(******************************************************************************************************************************************)
(****************************				           Reset Function Part                                                 *****************************)
(******************************************************************************************************************************************)
IF xReset THEN
	xReset:=FALSE;
	xSetEnd:=TRUE;
END_IF;
(******************************************************************************************************************************************)
(****************************				              Error Controlling Part                                            *****************************)
(******************************************************************************************************************************************)
IF (xSetError OR T_Station.TControl.xError) AND NOT(xSetEnd) THEN
	IF NOT(xInitError) THEN
		iStepError:=100;
		xInitError:=TRUE;
		T_Station.TControl.iCountDownPlungeCycle:=1;
		IF NOT(xSetError) THEN
			xSetError:=TRUE;
			xSetTmpError:=FALSE;
		ELSE
			xSetTmpError:=TRUE;
		END_IF;
	END_IF;
	CASE iStepError OF
		100:	IF T_Station.TControl.xError THEN
				diErrorNr:=T_Station.TControl.diErrorNr;
			END_IF;
			IF xSetTmpError THEN
				diErrorNr:=diTmpErrNr;
			END_IF;
			iStepError:=200;
		200:	IF xSetTmpError THEN
				xSetTmpError:=FALSE;
				xStopFctStation1:=FALSE;
				iStepError:=300;
			ELSE
				IF NOT(T_Station.TControl.xError) AND NOT(T_Station.TControl.xEnd) THEN
					IF (T_Station.TControl.iFunctNr = 1) THEN
						T_Station.TControl.xStop:=TRUE;
						xStopFctStation1:=TRUE;
					ELSE
						xStopFctStation1:=FALSE;
					END_IF;
				END_IF;
				iStepError:=300;
			END_IF;
		300:	IF xStopFctStation1 THEN
				IF NOT(T_Station.TControl.xStop) THEN
					xStopFctStation1:=FALSE;
				END_IF;
			END_IF;
			IF NOT(xStopFctStation1) THEN
				xError:=TRUE;
				iStepError:=400;
			END_IF;
		400:	IF xQuitErr THEN
				T_Station.TControl.xQuitError:=T_Station.TControl.xError;
				iStepError:=500;
			END_IF;
		500: IF NOT(T_Station.TControl.xQuitError) THEN
				xSetEnd:=TRUE;
			END_IF;
	END_CASE;
END_IF;
(******************************************************************************************************************************************)
(****************************				              Main Controlling Part                                            *****************************)
(******************************************************************************************************************************************)
IF (xStart OR xStartMainCtr) AND NOT(xSetEnd) AND NOT(xSetError) THEN
	IF NOT (xInitMainCtr) THEN
		iStepPrc:=10;
		xInitMainCtr:=TRUE;
		xStartMainCtr:=TRUE;
		xStart:=FALSE;
		xEnd:=FALSE;
		xSetEndPrc:=FALSE;
		iTmpFunctionNr:=1;
		xAbord:=FALSE;
		xProcessHold:=FALSE;
		T_ExchgParam.T_InfoValueCommon.iCountDownCycle:=1;
		xDoNotMovePositionOfToolFeeder:=FALSE;
		T_ExchgParam.T_InfoValueCommon.rActualWireFeedPosition:=0.0;
		T_ExchgParam.T_InfoValueCommon.rActualWireFeedSpeed:=0.0;
		(*08.07.2014: KFS	{	*)
		xWarmUp:= xWarmUpCycle:= T_ExchgParam.T_StationCommon.T_AutoGeometryPara.xWarmUp;
		xWarmUpDone:=FALSE;
		(*08.07.2014: KFS	}	*)
	END_IF;
	IF (xStopCycle AND NOT(xTmpStopCycle)) THEN
		IF (T_NovRAMData.T_ProcessImageData.T_AutoGeometryPara.iCycleGeometry <= 1) THEN
			xStopCycle:=xProcessHold:=FALSE;
			RETURN;
		END_IF;
		IF (iStepPrc = 40) AND NOT(xInitStep) THEN
			xTmpStopCycle:=TRUE;
		END_IF;
	END_IF;
	IF xTmpStopCycle THEN
		xStopCycle:=FALSE;
		xProcessHold:=TRUE;
		xTmpStopCycle:=FALSE;
		xInitStep:=xStartMainPrc:=FALSE;
		(*08.07.2014: KFS	{	*)
		xWarmUp:=FALSE;
		(*08.07.2014: KFS	}	*)
		iStepPrc:=100;
		RETURN;
	END_IF;
	IF xStop AND NOT(xTmpStop) THEN
		xTmpStop:=TRUE;
		iStepStop:=1;
	END_IF;
	IF xTmpStop THEN
		CASE iStepStop OF
		1:	IF NOT(T_Station.TControl.xEnd) THEN
				T_Station.TControl.xStop:=TRUE;
				iStepStop:=10;
			ELSE
				iStepStop:=20;
			END_IF;
		10:	IF NOT(T_Station.TControl.xStop) THEN
				iStepStop:=20;
			END_IF;
		20:	IF NOT(T_Station.TControl.xStart) AND T_Station.TControl.xEnd THEN
				T_Station.TControl.iFunctNr:=4;
				T_Station.TControl.xStart:=TRUE;
				T_Station.THardware.TAxisGrindFeeder.T_CtrleSingle.lrAcceleration:=T_NovRAMData.T_Standard.T_TeachINGrindFeeder.rAcceleration;
				T_Station.THardware.TAxisGrindFeeder.T_CtrleSingle.lrDecceleration:=T_NovRAMData.T_Standard.T_TeachINGrindFeeder.rDeceleration;
				T_Station.THardware.TAxisGrindFeeder.T_CtrleSingle.lrPosition:=	T_NovRAMData.T_ProcessImageData.T_ProcessPara.rToolDiameterProcess +
																			T_NovRAMData.T_ProcessImageData.T_ProcessPara.rSecurityPosGrindFeedProcess;
				T_Station.THardware.TAxisGrindFeeder.T_CtrleSingle.lrVelocity:=T_NovRAMData.T_ProcessImageData.T_ProcessPara.rSpeedBackwardGrindFeed;
				iStepStop:=30;
			END_IF;
		(* Check Active Movement of the Axis *)
		30:	IF NOT(T_Station.TControl.xStart) AND T_Station.TControl.xEnd THEN
				T_Station.TControl.iFunctNr:=18;	(* Check Axis Movement, and stop it if moves *)
				T_Station.TControl.xStart:=TRUE;
				iStepStop:=40;
			END_IF;
		40:	IF NOT(T_Station.TControl.xStart) AND T_Station.TControl.xEnd THEN
(*08.07.2014: KFS	{	*)
				IF iStepPrc = 105 THEN
					T_Station.THardware.TCylToolTension.T_CtrleCyl.iFunction:=2;
					T_Station.THardware.TCylToolTension.T_CtrleCyl.T_AnalogCylinder.rForceIn:=T_NovRAMData.T_ProcessImageData.T_ProcessPara.rToolTensionProcess;
					T_Station.THardware.TCylToolTension.T_Config.tDelayOn:=T#1s;
					T_Station.THardware.TCylToolTension.T_CtrleCyl.xExecute:=TRUE;
					T_Station.THardware.TCylToolLeftActive.T_CtrleCyl.iFunction:= 1;
					T_Station.THardware.TCylToolLeftActive.T_CtrleCyl.xExecute:=TRUE;
					T_Station.THardware.TCylToolRightActive.T_CtrleCyl.iFunction:=1;
					T_Station.THardware.TCylToolRightActive.T_CtrleCyl.xExecute:=TRUE;
					T_Station.THardware.TCylToolCenterActive.T_CtrleCyl.iFunction:=1;
					T_Station.THardware.TCylToolCenterActive.T_CtrleCyl.xExecute:=TRUE;
					T_Station.THardware.TCylToolPrismaLeftActive.T_CtrleCyl.iFunction:=1;
					T_Station.THardware.TCylToolPrismaLeftActive.T_CtrleCyl.xExecute:=TRUE;
					T_Station.THardware.TCylToolPrismaRightActive.T_CtrleCyl.iFunction:=1;
					T_Station.THardware.TCylToolPrismaRightActive.T_CtrleCyl.xExecute:=TRUE;
					iStepStop:=45;
				ELSE
(*08.07.2014: KFS	}	*)
					xStartMainPrc:=FALSE;
					xInitStep:=FALSE;
					iStepPrc:=0;
					xSetEnd:=TRUE;
					RETURN;
				END_IF
			END_IF;
		45:IF    (NOT(T_Station.THardware.TCylToolTension.T_CtrleCyl.xExecute) AND T_Station.THardware.TCylToolTension.T_CtrleCyl.xDone ) AND
		             (NOT(T_Station.THardware.TCylToolLeftActive.T_CtrleCyl.xExecute) AND T_Station.THardware.TCylToolLeftActive.T_CtrleCyl.xDone ) AND
			    (NOT(T_Station.THardware.TCylToolRightActive.T_CtrleCyl.xExecute) AND T_Station.THardware.TCylToolRightActive.T_CtrleCyl.xDone ) AND
			    (NOT(T_Station.THardware.TCylToolCenterActive.T_CtrleCyl.xExecute) AND T_Station.THardware.TCylToolCenterActive.T_CtrleCyl.xDone ) AND
			    (NOT(T_Station.THardware.TCylToolPrismaLeftActive.T_CtrleCyl.xExecute) AND T_Station.THardware.TCylToolPrismaLeftActive.T_CtrleCyl.xDone ) AND
			    (NOT(T_Station.THardware.TCylToolPrismaRightActive.T_CtrleCyl.xExecute) AND T_Station.THardware.TCylToolPrismaRightActive.T_CtrleCyl.xDone )		THEN
				xStartMainPrc:=FALSE;
				xInitStep:=FALSE;
				iStepPrc:=0;
				xSetEnd:=TRUE;
				RETURN;
			END_IF;
		END_CASE;
		RETURN;
	END_IF;
	IF NOT(xStartMainPrc) THEN
		xStartMainPrc:=TRUE;
	END_IF;
END_IF;
(******************************************************************************************************************************************)
(****************************				             Main Procedure Part                                             *****************************)
(******************************************************************************************************************************************)
(*08.07.2014: KFS	{	*)
IF xWarmUp AND NOT(xWarmUpDone)THEN
	TONWarmUpTimer(IN:=TRUE,PT:=T#45m);
	IF TONWarmUpTimer.Q THEN
		TONWarmUpTimer(IN:=FALSE);
		xWarmUpDone:=TRUE;
	END_IF;
ELSE
	TONWarmUpTimer(IN:=FALSE);
END_IF;
(*08.07.2014: KFS	}	*)
IF xStartProcess THEN
	TONStartTimer(IN:=TRUE,PT:=T#1s);
	IF TONStartTimer.Q THEN
		TONStartTimer(IN:=FALSE);
		IF (T_ExchgParam.T_InfoValueCommon.tAutoTimeLeft >= T#1s) THEN
			T_ExchgParam.T_InfoValueCommon.tAutoTimeLeft:=T_ExchgParam.T_InfoValueCommon.tAutoTimeLeft - T#1s;
		ELSE
			T_ExchgParam.T_InfoValueCommon.tAutoTimeLeft:=T#0s;
		END_IF;
	END_IF;
	tStepTime:=T_ExchgParam.T_InfoValueCommon.tAutoTimeTotal / 100;
	TONStartTimer1(IN:=TRUE,PT:=tStepTime);
	IF TONStartTimer1.Q THEN
		TONStartTimer1(IN:=FALSE);
		T_ExchgParam.T_InfoValueCommon.bProgressbarAutoGeometry:=T_ExchgParam.T_InfoValueCommon.bProgressbarAutoGeometry + 1;
		IF (T_ExchgParam.T_InfoValueCommon.bProgressbarAutoGeometry >= 100) THEN
			T_ExchgParam.T_InfoValueCommon.bProgressbarAutoGeometry:=100;
		END_IF;
	END_IF;
ELSE
	TONStartTimer(IN:=FALSE);
	TONStartTimer1(IN:=FALSE);
END_IF;
IF xStartMainPrc AND NOT(xSetEnd) AND NOT(xSetError) THEN
	CASE iStepPrc OF
		(* Check first if the AutoGeometry is available to start it *)
		10:	T_Station.THardware.TAxisToolLeft.T_CtrleSingle.lrAcceleration:=T_NovRAMData.T_Standard.T_TeachINToolLeft.rAcceleration;
			T_Station.THardware.TAxisToolLeft.T_CtrleSingle.lrDecceleration:=T_NovRAMData.T_Standard.T_TeachINToolLeft.rDeceleration;
			T_Station.THardware.TAxisToolCenter.T_CtrleSingle.lrAcceleration:=T_NovRAMData.T_Standard.T_TeachINToolCenter.rAcceleration;
			T_Station.THardware.TAxisToolCenter.T_CtrleSingle.lrDecceleration:=T_NovRAMData.T_Standard.T_TeachINToolCenter.rDeceleration;
			T_Station.THardware.TAxisToolRight.T_CtrleSingle.lrAcceleration:=T_NovRAMData.T_Standard.T_TeachINToolRight.rAcceleration;
			T_Station.THardware.TAxisToolRight.T_CtrleSingle.lrDecceleration:=T_NovRAMData.T_Standard.T_TeachINToolRight.rDeceleration;
			T_Station.THardware.TAxisToolFeeder.T_CtrleSingle.lrAcceleration:=T_NovRAMData.T_Standard.T_TeachINToolFeeder.rAcceleration;
			T_Station.THardware.TAxisToolFeeder.T_CtrleSingle.lrDecceleration:=T_NovRAMData.T_Standard.T_TeachINToolFeeder.rDeceleration;
			T_Station.THardware.TAxisGrindFeeder.T_CtrleSingle.lrAcceleration:=T_NovRAMData.T_Standard.T_TeachINGrindFeeder.rAcceleration;
			T_Station.THardware.TAxisGrindFeeder.T_CtrleSingle.lrDecceleration:=T_NovRAMData.T_Standard.T_TeachINGrindFeeder.rDeceleration;
			(* Only for MicroRod, check if the tool is clamped *)
			IF xMicroRodActive THEN
				(*22.12.2009: KFS	{ *)
				(*Added control if all cylinder for the tool are activated*)
				IF ( T_Station.THardware.TCylToolTension.T_CtrleCyl.xStatePosOn AND NOT( xWarmUp) )OR
				    T_Station.THardware.TCylToolLeftActive.T_CtrleCyl.T_Standard.xActivOn OR
 				    T_Station.THardware.TCylToolRightActive.T_CtrleCyl.T_Standard.xActivOn OR
				   (* T_Station.THardware.TCylToolCenterActive.T_CtrleCyl.T_Standard.xActivOn OR*)	(* IGS auskommentiert, diesen Zyl gibts auf der M3 nicht *)
				   ( NOT(T_Station.THardware.TCylToolPrismaLeftActive.T_CtrleCyl.T_Standard.xActivOn) AND NOT(xWarmUp)) OR
				   ( NOT(T_Station.THardware.TCylToolPrismaRightActive.T_CtrleCyl.T_Standard.xActivOn) AND NOT(xWarmUp))  	THEN
						xSetError:=TRUE;
						diTmpErrNr:=2;			(* Tool is not clamped *)
				END_IF;
				(*22.12.2009: KFS	} *)
			END_IF;
			(* Only for MicroRod, check if the Machine is referenced *)
			IF xMicroRodActive THEN
				IF NOT(T_Station.TControl.xReferenced) THEN
					xSetError:=TRUE;
					diTmpErrNr:=1;	(* Machine is not referenced *)
					RETURN;
				END_IF;
			END_IF;
			xStartMainPrc:=FALSE;
			xInitStep:=FALSE;
			iStepPrc:=11;
		(* Set the ToolTension force *)
		11:	IF NOT(xInitStep) THEN
				xInitStep:=TRUE;
				T_Station.THardware.TCylToolTension.T_CtrleCyl.iFunction:=2;	(* activate the ToolTension *)
				T_Station.THardware.TCylToolTension.T_CtrleCyl.T_AnalogCylinder.rForceIn:=T_NovRAMData.T_ProcessImageData.T_ProcessPara.rToolTensionProcess;
				IF xMicroRodActive THEN
					T_Station.THardware.TCylToolTension.T_Config.tDelayOn:=T#1s;
				ELSE
					T_Station.THardware.TCylToolTension.T_Config.tDelayOn:=T#0s;
				END_IF;
				T_Station.THardware.TCylToolTension.T_CtrleCyl.xExecute:=TRUE;
			END_IF;
			IF NOT(T_Station.THardware.TCylToolTension.T_CtrleCyl.xExecute) AND T_Station.THardware.TCylToolTension.T_CtrleCyl.xDone THEN
				(* Only for MicroRod, check if the tool is clamped *)
				IF xMicroRodActive THEN
					IF T_Station.THardware.TCylToolTension.T_CtrleCyl.xStatePosOn AND NOT( xWarmUp) THEN
						xSetError:=TRUE;
						diTmpErrNr:=2;			(* Tool is not clamped *)
						RETURN;
					END_IF;
				END_IF;
				iStepPrc:=20;
				xStartMainPrc:=FALSE;
				xInitStep:=FALSE;
			END_IF;
		(* Switch First all Axis the power supply on *)
		20:	IF NOT(xInitStep) THEN
				xInitStep:=TRUE;
				T_Station.TControl.iFunctNr:=16;
				T_Station.TControl.xStart:=TRUE;
			END_IF;
			IF NOT(T_Station.TControl.xStart) AND T_Station.TControl.xEnd THEN
				iStepPrc:=30;
				xStartMainPrc:=FALSE;
				xInitStep:=FALSE;
				iTmpStationFunctionNr:=6;
				T_Station.THardware.TAxisToolLeft.T_CtrleSingle.rSetPosition:=0.0;
				T_Station.THardware.TAxisToolCenter.T_CtrleSingle.rSetPosition:=0.0;
				T_Station.THardware.TAxisToolRight.T_CtrleSingle.rSetPosition:=0.0;
				T_Station.THardware.TAxisToolFeeder.T_CtrleSingle.rSetPosition:=0.0;
			END_IF;
		(* Reset the Position of the Axis *)
		30:	IF NOT(xInitStep) THEN
				xInitStep:=TRUE;
				(* 6=ToolLeft, 7=ToolCenter, 8=ToolRight, 9=ToolFeeder *)
				T_Station.TControl.iFunctNr:=iTmpStationFunctionNr;
				T_Station.TControl.xStart:=TRUE;
			END_IF;
			IF NOT(T_Station.TControl.xStart) AND T_Station.TControl.xEnd THEN
				iTmpStationFunctionNr:=iTmpStationFunctionNr + 1;
				IF NOT(xMicroRodActive) AND (iTmpStationFunctionNr = 7) THEN
					iTmpStationFunctionNr:=iTmpStationFunctionNr + 1;
				END_IF;
				IF xMicroRodActive AND (iTmpStationFunctionNr = 9) THEN
					iTmpStationFunctionNr:=iTmpStationFunctionNr + 1;
				END_IF;
				xStartMainPrc:=FALSE;
				xInitStep:=FALSE;
				IF (iTmpStationFunctionNr < 10) THEN
					iStepPrc:=30;
				ELSE
					iStepPrc:=40;
				END_IF;
			END_IF;
		(* GrindFeeder Set Absolut to Security Position *)
		40:	IF NOT(xInitStep) THEN
				xInitStep:=TRUE;
				T_Station.TControl.iFunctNr:=4;
				T_Station.TControl.xStart:=TRUE;
				T_Station.THardware.TAxisGrindFeeder.T_CtrleSingle.lrAcceleration:=T_NovRAMData.T_Standard.T_TeachINGrindFeeder.rAcceleration;
				T_Station.THardware.TAxisGrindFeeder.T_CtrleSingle.lrDecceleration:=T_NovRAMData.T_Standard.T_TeachINGrindFeeder.rDeceleration;
				T_Station.THardware.TAxisGrindFeeder.T_CtrleSingle.lrPosition:=	T_NovRAMData.T_ProcessImageData.T_ProcessPara.rToolDiameterProcess +
																			T_NovRAMData.T_ProcessImageData.T_ProcessPara.rSecurityPosGrindFeedProcess;
				T_Station.THardware.TAxisGrindFeeder.T_CtrleSingle.lrVelocity:=T_NovRAMData.T_ProcessImageData.T_ProcessPara.rSpeedBackwardGrindFeed;
			END_IF;
			IF NOT(T_Station.TControl.xStart) AND T_Station.TControl.xEnd THEN
				IF xMicroRodActive THEN
					IF xDoNotMovePositionOfToolFeeder THEN
						iStepPrc:=60;
					ELSE
						iStepPrc:=50;
					END_IF;
				ELSE
					iStepPrc:=60;
				END_IF;
				xStartMainPrc:=FALSE;
				xInitStep:=FALSE;
			END_IF;
		(* Only for MicroRod-->Set ToolFeed Absolut to the Zero Position*)
		50:	IF NOT(xInitStep) THEN
(* 04.04.2011: KFS	{ 	Neu wird die Längeneinstellung des ToolFeeders nicht mehr kontrolliert und direkt auf die StartPos gefahren(vormals RefPos)!
				xInitStep:=TRUE;
				T_Station.TControl.iFunctNr:=14;
				T_Station.TControl.xStart:=TRUE;
				T_Station.THardware.TAxisToolFeeder.T_CtrleSingle.lrAcceleration:=T_NovRAMData.T_Standard.T_TeachINToolFeeder.rAcceleration;
				T_Station.THardware.TAxisToolFeeder.T_CtrleSingle.lrDecceleration:=T_NovRAMData.T_Standard.T_TeachINToolFeeder.rDeceleration;
				T_Station.THardware.TAxisToolFeeder.T_CtrleSingle.lrPosition:=0.0;
				T_Station.THardware.TAxisToolFeeder.T_CtrleSingle.lrVelocity:=T_NovRAMData.T_ProcessImageData.T_ProcessPara.rSpeedStartPosToolFeedProcess;
			END_IF;
			IF NOT(T_Station.TControl.xStart) AND T_Station.TControl.xEnd THEN
 04.04.2011: KFS	}	*)
				(*30.09.2010: KFS	{ *)
				(* Check first settled geometry parameter *)
				FBCheckToolGeometryPara(	iProcessNr:= 1,
											T_GeometryCommon:= T_ExchgParam.T_GeometryCommon,
											T_AutoGeometryPara:= T_NovRAMData.T_ProcessImageData.T_AutoGeometryPara,
											T_AutoGroovePara:= T_NovRAMData.T_ProcessImageData.T_AutoGroovePara,
											T_ProcessPara:= T_NovRamData.T_ProcessImageData.T_ProcessPara,
											rToolDiameter:=T_NovRAMData.T_ProcessImageData.T_ProcessPara.rToolDiameterProcess,
											xMicroRodActive:=xMicroRodActive,
											(*rOffsetMaxToolLength:= T_Station.THardware.TToolFeederWorkLength.T_CtrleCyl.T_Analog.rLengthIn*));
				IF FBCheckToolGeometryPara.xError THEN
					xSetError:=TRUE;
					diTmpErrNr:=FBCheckToolGeometryPara.diErrorNr;
					RETURN;
				END_IF;
				(*30.09.2010: KFS	} *)
				iStepPrc:=55;
				xStartMainPrc:=FALSE;
				xInitStep:=FALSE;
			END_IF;
		(* Only for MicroRod-->Set ToolFeed Absolut to the StartPosition and if more cycle than only the first time *)
		55:	IF NOT(xInitStep) THEN
				xInitStep:=TRUE;
				T_Station.TControl.iFunctNr:=14;
				T_Station.TControl.xStart:=TRUE;
				T_Station.THardware.TAxisToolFeeder.T_CtrleSingle.lrAcceleration:=T_NovRAMData.T_Standard.T_TeachINToolFeeder.rAcceleration;
				T_Station.THardware.TAxisToolFeeder.T_CtrleSingle.lrDecceleration:=T_NovRAMData.T_Standard.T_TeachINToolFeeder.rDeceleration;
				T_Station.THardware.TAxisToolFeeder.T_CtrleSingle.lrPosition:=T_NovRAMData.T_ProcessImageData.T_ProcessPara.rStartPosToolFeedAuto;
				T_Station.THardware.TAxisToolFeeder.T_CtrleSingle.lrVelocity:=T_NovRAMData.T_ProcessImageData.T_ProcessPara.rSpeedStartPosToolFeedProcess;
			END_IF;
			IF NOT(T_Station.TControl.xStart) AND T_Station.TControl.xEnd THEN
				iStepPrc:=60;
				xStartMainPrc:=FALSE;
				xInitStep:=FALSE;
			END_IF;
		(* ToolRotation Start *)
		60:	IF NOT(xInitStep) THEN
				xInitStep:=TRUE;
				T_Station.TControl.iFunctNr:=2;
				T_Station.TControl.xStart:=TRUE;
				(* ToolLeft --> Master *)
				T_Station.THardware.TAxisToolLeft.T_CtrleSingle.lrVelocity:=T_NovRAMData.T_ProcessImageData.T_AutoGeometryPara.rSpeedToolRotationGeometry;
				T_Station.THardware.TAxisToolLeft.T_CtrleSingle.lrAcceleration:=T_NovRAMData.T_Standard.T_TeachINToolLeft.rAcceleration;
				T_Station.THardware.TAxisToolLeft.T_CtrleSingle.lrDecceleration:=T_NovRAMData.T_Standard.T_TeachINToolLeft.rDeceleration;
				IF xMicroRodActive THEN
					(* ToolCenter --> Slave of ToolLeft only by MicroRod *)
					T_Station.THardware.TAxisToolCenter.T_CtrleSingle.lrAcceleration:=T_NovRAMData.T_Standard.T_TeachINToolCenter.rAcceleration;
					T_Station.THardware.TAxisToolCenter.T_CtrleSingle.lrDecceleration:=T_NovRAMData.T_Standard.T_TeachINToolCenter.rDeceleration;
					T_Station.THardware.TAxisToolCenter.T_CtrleSingle.lrGearDivider:=INT_TO_LREAL(T_Station.T_WorkTool.iBaseGearDivider);
					T_Station.THardware.TAxisToolCenter.T_CtrleSingle.lrGearFactor:=(	INT_TO_LREAL(T_Station.T_WorkTool.iBaseGearDivider) /
																					(T_Station.THardware.TAxisToolLeft.T_CtrleSingle.lrGearRatio /
																					T_Station.THardware.TAxisToolCenter.T_CtrleSingle.lrGearRatio)) * -1.0;

					(* ToolRight --> Slave of ToolLeft by MicroWire or Slave of ToolRight by MicroRod *)
					T_Station.THardware.TAxisToolRight.T_CtrleSingle.lrAcceleration:=T_NovRAMData.T_Standard.T_TeachINToolRight.rAcceleration;
					T_Station.THardware.TAxisToolRight.T_CtrleSingle.lrDecceleration:=T_NovRAMData.T_Standard.T_TeachINToolRight.rDeceleration;
					T_Station.THardware.TAxisToolRight.T_CtrleSingle.lrGearDivider:=INT_TO_LREAL(T_Station.T_WorkTool.iBaseGearDivider);
					T_Station.THardware.TAxisToolRight.T_CtrleSingle.lrGearFactor:=	INT_TO_LREAL(T_Station.T_WorkTool.iBaseGearDivider) /
																					(T_Station.THardware.TAxisToolLeft.T_CtrleSingle.lrGearRatio /
		 																			T_Station.THardware.TAxisToolRight.T_CtrleSingle.lrGearRatio);
				END_IF;
				IF NOT(xMicroRodActive) THEN
					(* ToolRight --> Slave of ToolRight by MicroWire *)
					T_Station.THardware.TAxisToolFeeder.T_CtrleSingle.lrAcceleration:=T_NovRAMData.T_Standard.T_TeachINToolFeeder.rAcceleration;
					T_Station.THardware.TAxisToolFeeder.T_CtrleSingle.lrDecceleration:=T_NovRAMData.T_Standard.T_TeachINToolFeeder.rDeceleration;
					T_Station.THardware.TAxisToolFeeder.T_CtrleSingle.lrGearDivider:=INT_TO_LREAL(T_Station.T_WorkTool.iBaseGearDivider);
					T_Station.THardware.TAxisToolFeeder.T_CtrleSingle.lrGearFactor:=	(INT_TO_LREAL(T_Station.T_WorkTool.iBaseGearDivider) /
																					(T_Station.THardware.TAxisToolFeeder.T_CtrleSingle.lrGearRatio /
																					T_Station.THardware.TAxisToolRight.T_CtrleSingle.lrGearRatio)) * -1.0;

					(* ToolRight --> Slave of ToolLeft by MicroWire or Slave of ToolRight by MicroRod *)
					T_Station.THardware.TAxisToolRight.T_CtrleSingle.lrAcceleration:=T_NovRAMData.T_Standard.T_TeachINToolRight.rAcceleration;
					T_Station.THardware.TAxisToolRight.T_CtrleSingle.lrDecceleration:=T_NovRAMData.T_Standard.T_TeachINToolRight.rDeceleration;
					T_Station.THardware.TAxisToolRight.T_CtrleSingle.lrGearDivider:=INT_TO_LREAL(T_Station.T_WorkTool.iBaseGearDivider);
					T_Station.THardware.TAxisToolRight.T_CtrleSingle.lrGearFactor:=	(INT_TO_LREAL(T_Station.T_WorkTool.iBaseGearDivider) /
																					(T_Station.THardware.TAxisToolLeft.T_CtrleSingle.lrGearRatio /
																					T_Station.THardware.TAxisToolRight.T_CtrleSingle.lrGearRatio)) * -1.0;
				END_IF;
			END_IF;
			IF NOT(T_Station.TControl.xStart) AND T_Station.TControl.xEnd THEN
				xStartMainPrc:=FALSE;
				xInitStep:=FALSE;
				iStepPrc:=70;
			END_IF;
		(* GrindFeeder Set Absolut to ToolDiameter minus the offset with the fast speed *)
		70:  	IF NOT(xInitStep) THEN
				xInitStep:=TRUE;
				T_Station.TControl.iFunctNr:=4;
				T_Station.TControl.xStart:=TRUE;
				T_Station.THardware.TAxisGrindFeeder.T_CtrleSingle.lrAcceleration:=T_NovRAMData.T_Standard.T_TeachINGrindFeeder.rAcceleration;
				T_Station.THardware.TAxisGrindFeeder.T_CtrleSingle.lrDecceleration:=T_NovRAMData.T_Standard.T_TeachINGrindFeeder.rDeceleration;
				T_Station.THardware.TAxisGrindFeeder.T_CtrleSingle.lrPosition:=T_NovRAMData.T_ProcessImageData.T_ProcessPara.rToolDiameterProcess + T_NovRAMData.T_ProcessImageData.T_ProcessPara.rOffsetBeforeToolDiaGrindFeedProcess;
				T_Station.THardware.TAxisGrindFeeder.T_CtrleSingle.lrVelocity:=T_NovRAMData.T_ProcessImageData.T_ProcessPara.rSpeedForwardFastGrindFeed;
			END_IF;
			IF NOT(T_Station.TControl.xStart) AND T_Station.TControl.xEnd THEN
				xStartMainPrc:=FALSE;
				xInitStep:=FALSE;
				iStepPrc:=80;
			END_IF;
		(* Working AutoGeometry *)
		80:	IF NOT(xInitStep) THEN
				xStartProcess:=TRUE;
				xInitStep:=TRUE;
				T_Station.TControl.iFunctNr:=19;
				T_Station.TControl.xStart:=TRUE;
			END_IF;
			IF NOT(T_Station.TControl.xStart) AND T_Station.TControl.xEnd THEN
				xStartMainPrc:=FALSE;
				xInitStep:=FALSE;
				iStepPrc:=90;
				RETURN;
			END_IF;
			(* Only for MicroRod, check if the tool is clamped *)
			IF xMicroRodActive THEN
				IF T_Station.THardware.TCylToolTension.T_CtrleCyl.xStatePosOn AND NOT( xWarmUp) THEN
					xStartMainPrc:=FALSE;
					xInitStep:=FALSE;
					iStepPrc:=81;
					RETURN;
				END_IF;
			END_IF;
			T_ExchgParam.T_InfoValueCommon.iCountDownPlungeCycle:=T_Station.TControl.iCountDownPlungeCycle;
		(* Stop the Process, because the Tool is broken *)
		81:	IF NOT(xInitStep) THEN
				xInitStep:=TRUE;
				T_Station.TControl.xStop:=TRUE;
			END_IF;
			IF NOT(T_Station.TControl.xStart) AND T_Station.TControl.xEnd THEN
				xStartMainPrc:=FALSE;
				xInitStep:=FALSE;
				iStepPrc:=82;
			END_IF;
		(* Set the GrindFeeder to the security Position *)
		82:	IF NOT(xInitStep) THEN
				xInitStep:=TRUE;
				T_Station.TControl.iFunctNr:=4;
				T_Station.TControl.xStart:=TRUE;
				T_Station.THardware.TAxisGrindFeeder.T_CtrleSingle.lrAcceleration:=T_NovRAMData.T_Standard.T_TeachINGrindFeeder.rAcceleration;
				T_Station.THardware.TAxisGrindFeeder.T_CtrleSingle.lrDecceleration:=T_NovRAMData.T_Standard.T_TeachINGrindFeeder.rDeceleration;
				T_Station.THardware.TAxisGrindFeeder.T_CtrleSingle.lrPosition:=	T_NovRAMData.T_ProcessImageData.T_ProcessPara.rToolDiameterProcess +
																			T_NovRAMData.T_ProcessImageData.T_ProcessPara.rSecurityPosGrindFeedProcess;
				T_Station.THardware.TAxisGrindFeeder.T_CtrleSingle.lrVelocity:=T_NovRAMData.T_ProcessImageData.T_ProcessPara.rSpeedBackwardGrindFeed;
			END_IF;
			IF NOT(T_Station.TControl.xStart) AND T_Station.TControl.xEnd THEN
				xStartMainPrc:=FALSE;
				xInitStep:=FALSE;
				iStepPrc:=83;
			END_IF;
		(* Check Active Movement of the Axis *)
		83:	IF NOT(xInitStep) THEN
				xInitStep:=TRUE;
				T_Station.TControl.iFunctNr:=18;	(* Check Axis Movement, and stop it if moves *)
				T_Station.TControl.xStart:=TRUE;
			END_IF;
			IF NOT(T_Station.TControl.xStart) AND T_Station.TControl.xEnd THEN
				xSetError:=TRUE;
				diTmpErrNr:=2;			(* Tool is not clamped *)
				RETURN;
			END_IF;
		(* GrindFeeder Set Absolut to Security Position *)
		90:	IF NOT(xInitStep) THEN
				xInitStep:=TRUE;
				T_Station.TControl.iFunctNr:=4;
				T_Station.TControl.xStart:=TRUE;
				T_Station.THardware.TAxisGrindFeeder.T_CtrleSingle.lrAcceleration:=T_NovRAMData.T_Standard.T_TeachINGrindFeeder.rAcceleration;
				T_Station.THardware.TAxisGrindFeeder.T_CtrleSingle.lrDecceleration:=T_NovRAMData.T_Standard.T_TeachINGrindFeeder.rDeceleration;
				T_Station.THardware.TAxisGrindFeeder.T_CtrleSingle.lrPosition:=	T_NovRAMData.T_ProcessImageData.T_ProcessPara.rToolDiameterProcess +
																			T_NovRAMData.T_ProcessImageData.T_ProcessPara.rSecurityPosGrindFeedProcess;
				T_Station.THardware.TAxisGrindFeeder.T_CtrleSingle.lrVelocity:=T_NovRAMData.T_ProcessImageData.T_ProcessPara.rSpeedBackwardGrindFeed;
				T_ExchgParam.T_StationCommon.T_AutoGeometryPara.xMoveTableStuderBW:=TRUE; (*SOA*)
				TONWaitForTableMovement(IN:=TRUE,PT:=T#2s);
			END_IF;
			IF NOT(T_Station.TControl.xStart) AND T_Station.TControl.xEnd THEN
				xStartMainPrc:=FALSE;
				xInitStep:=FALSE;
				IF (T_NovRAMData.T_ProcessImageData.T_AutoGeometryPara.iCycleGeometry > T_ExchgParam.T_InfoValueCommon.iCountDownCycle) THEN
					IF NOT(xStopCycle) THEN
						T_ExchgParam.T_InfoValueCommon.iCountDownCycle:=T_ExchgParam.T_InfoValueCommon.iCountDownCycle + 1;
					END_IF;
					xDoNotMovePositionOfToolFeeder:=TRUE;
					iStepPrc:=40;	(* Repeat to work the same Geometry *)
				ELSE
					IF TONWaitForTableMovement.Q THEN
						TONWaitForTableMovement.IN:=FALSE;
						iStepPrc:=100;
					END_IF
				END_IF;
			END_IF;
		(* ToolRotation Stop *)
		100:	IF NOT(xInitStep) THEN
				xInitStep:=TRUE;
				T_Station.TControl.iFunctNr:=3;
				T_Station.TControl.xStart:=TRUE;
				(* ToolLeft --> Master *)
				T_Station.THardware.TAxisToolLeft.T_CtrleSingle.lrAcceleration:=T_NovRAMData.T_Standard.T_TeachINToolLeft.rAcceleration;
				T_Station.THardware.TAxisToolLeft.T_CtrleSingle.lrDecceleration:=T_NovRAMData.T_Standard.T_TeachINToolLeft.rDeceleration;
				IF xMicroRodActive THEN
					(* ToolCenter --> Slave of ToolLeft only by MicroRod *)
					T_Station.THardware.TAxisToolCenter.T_CtrleSingle.lrAcceleration:=T_NovRAMData.T_Standard.T_TeachINToolCenter.rAcceleration;
					T_Station.THardware.TAxisToolCenter.T_CtrleSingle.lrDecceleration:=T_NovRAMData.T_Standard.T_TeachINToolCenter.rDeceleration;
				END_IF;
				(* ToolRight --> Slave of ToolLeft by MicroWire or Slave of ToolRight by MicroRod *)
				T_Station.THardware.TAxisToolRight.T_CtrleSingle.lrAcceleration:=T_NovRAMData.T_Standard.T_TeachINToolRight.rAcceleration;
				T_Station.THardware.TAxisToolRight.T_CtrleSingle.lrDecceleration:=T_NovRAMData.T_Standard.T_TeachINToolRight.rDeceleration;
				IF NOT(xMicroRodActive) THEN
					(* ToolRight --> Slave of ToolRight by MicroWire *)
					T_Station.THardware.TAxisToolFeeder.T_CtrleSingle.lrAcceleration:=T_NovRAMData.T_Standard.T_TeachINToolFeeder.rAcceleration;
					T_Station.THardware.TAxisToolFeeder.T_CtrleSingle.lrDecceleration:=T_NovRAMData.T_Standard.T_TeachINToolFeeder.rDeceleration;
				END_IF;
			END_IF;
			IF NOT(T_Station.TControl.xStart) AND T_Station.TControl.xEnd THEN
				xStartMainPrc:=FALSE;
				xInitStep:=FALSE;
				IF NOT(xWarmUpCycle) THEN
					iStepPrc:=110;
				ELSE
					iStepPrc:=102;
				END_IF;
			END_IF;
(*08.07.2014: KFS	{	*)
		102:	IF NOT(xInitStep) THEN
				T_Station.THardware.TCylToolTension.T_CtrleCyl.iFunction:=1;
				T_Station.THardware.TCylToolTension.T_CtrleCyl.xExecute:=TRUE;
				T_Station.THardware.TCylToolLeftActive.T_CtrleCyl.iFunction:= 2;
				T_Station.THardware.TCylToolLeftActive.T_CtrleCyl.xExecute:=TRUE;
				T_Station.THardware.TCylToolRightActive.T_CtrleCyl.iFunction:=2;
				T_Station.THardware.TCylToolRightActive.T_CtrleCyl.xExecute:=TRUE;
				T_Station.THardware.TCylToolCenterActive.T_CtrleCyl.iFunction:=2;
				T_Station.THardware.TCylToolCenterActive.T_CtrleCyl.xExecute:=TRUE;
				T_Station.THardware.TCylToolPrismaLeftActive.T_CtrleCyl.iFunction:=51;
				T_Station.THardware.TCylToolPrismaLeftActive.T_CtrleCyl.xExecute:=TRUE;
				T_Station.THardware.TCylToolPrismaRightActive.T_CtrleCyl.iFunction:=51;
				T_Station.THardware.TCylToolPrismaRightActive.T_CtrleCyl.xExecute:=TRUE;
				xInitStep:=TRUE;
			END_IF;
			IF(NOT(T_Station.THardware.TCylToolTension.T_CtrleCyl.xExecute) AND T_Station.THardware.TCylToolTension.T_CtrleCyl.xDone ) AND
			    (NOT(T_Station.THardware.TCylToolLeftActive.T_CtrleCyl.xExecute) AND T_Station.THardware.TCylToolLeftActive.T_CtrleCyl.xDone ) AND
			    (NOT(T_Station.THardware.TCylToolRightActive.T_CtrleCyl.xExecute) AND T_Station.THardware.TCylToolRightActive.T_CtrleCyl.xDone ) AND
			    (NOT(T_Station.THardware.TCylToolCenterActive.T_CtrleCyl.xExecute) AND T_Station.THardware.TCylToolCenterActive.T_CtrleCyl.xDone ) AND
			    (NOT(T_Station.THardware.TCylToolPrismaLeftActive.T_CtrleCyl.xExecute) AND T_Station.THardware.TCylToolPrismaLeftActive.T_CtrleCyl.xDone ) AND
			    (NOT(T_Station.THardware.TCylToolPrismaRightActive.T_CtrleCyl.xExecute) AND T_Station.THardware.TCylToolPrismaRightActive.T_CtrleCyl.xDone )		THEN
				TONWarmUpBreakTimer(IN:=FALSE);
				xStartMainPrc:=FALSE;
				xInitStep:=FALSE;
				iStepPrc:=105;
			END_IF;
		105: IF xWarmUpDone THEN
				T_ExchgParam.T_StationCommon.T_AutoGeometryPara.xWarmUp:=FALSE;
			END_IF;
			TONWarmUpBreakTimer(IN:=TRUE,PT:=T#20s);
			IF TONWarmUpBreakTimer.Q THEN
				TONWarmUpBreakTimer(IN:=FALSE);
				T_ExchgParam.T_InfoValueCommon.iCountDownCycle:=1;
				xDoNotMovePositionOfToolFeeder:=FALSE;
				xStartMainPrc:=FALSE;
				xInitStep:=FALSE;
				iStepPrc:=107;
			END_IF;
		107:	IF NOT(xInitStep) THEN
				T_Station.THardware.TCylToolTension.T_CtrleCyl.iFunction:=2;
				T_Station.THardware.TCylToolTension.T_CtrleCyl.T_AnalogCylinder.rForceIn:=T_NovRAMData.T_ProcessImageData.T_ProcessPara.rToolTensionProcess;
				T_Station.THardware.TCylToolTension.T_Config.tDelayOn:=T#1s;
				T_Station.THardware.TCylToolTension.T_CtrleCyl.xExecute:=TRUE;
				T_Station.THardware.TCylToolLeftActive.T_CtrleCyl.iFunction:= 1;
				T_Station.THardware.TCylToolLeftActive.T_CtrleCyl.xExecute:=TRUE;
				T_Station.THardware.TCylToolRightActive.T_CtrleCyl.iFunction:=1;
				T_Station.THardware.TCylToolRightActive.T_CtrleCyl.xExecute:=TRUE;
				T_Station.THardware.TCylToolCenterActive.T_CtrleCyl.iFunction:=1;
				T_Station.THardware.TCylToolCenterActive.T_CtrleCyl.xExecute:=TRUE;
				T_Station.THardware.TCylToolPrismaLeftActive.T_CtrleCyl.iFunction:=51;
				T_Station.THardware.TCylToolPrismaLeftActive.T_CtrleCyl.xExecute:=TRUE;
				T_Station.THardware.TCylToolPrismaRightActive.T_CtrleCyl.iFunction:=51;
				T_Station.THardware.TCylToolPrismaRightActive.T_CtrleCyl.xExecute:=TRUE;
				xInitStep:=TRUE;
			END_IF;
			IF(NOT(T_Station.THardware.TCylToolTension.T_CtrleCyl.xExecute) AND T_Station.THardware.TCylToolTension.T_CtrleCyl.xDone ) AND
			    (NOT(T_Station.THardware.TCylToolLeftActive.T_CtrleCyl.xExecute) AND T_Station.THardware.TCylToolLeftActive.T_CtrleCyl.xDone ) AND
			    (NOT(T_Station.THardware.TCylToolRightActive.T_CtrleCyl.xExecute) AND T_Station.THardware.TCylToolRightActive.T_CtrleCyl.xDone ) AND
			    (NOT(T_Station.THardware.TCylToolCenterActive.T_CtrleCyl.xExecute) AND T_Station.THardware.TCylToolCenterActive.T_CtrleCyl.xDone ) AND
			    (NOT(T_Station.THardware.TCylToolPrismaLeftActive.T_CtrleCyl.xExecute) AND T_Station.THardware.TCylToolPrismaLeftActive.T_CtrleCyl.xDone ) AND
			    (NOT(T_Station.THardware.TCylToolPrismaRightActive.T_CtrleCyl.xExecute) AND T_Station.THardware.TCylToolPrismaRightActive.T_CtrleCyl.xDone )		THEN
				xStartMainPrc:=FALSE;
				xInitStep:=FALSE;
				iStepPrc:=10;
			END_IF;
(*08.07.2014: KFS	}	*)
		110:	xSetEndPrc:=FALSE;
			xStartMainPrc:=FALSE;
			xInitStep:=FALSE;
			iStepPrc:=0;
			xSetEnd:=TRUE;
	END_CASE;
END_IF;
(******************************************************************************************************************************************)
(****************************				             	Init / Reset Part                                                   *****************************)
(******************************************************************************************************************************************)
IF xSetEnd THEN
	xEnd:=TRUE;
	xInitStep:=FALSE;
	xSetEnd:=FALSE;
	xStop:=FALSE;
	xStopCycle:=FALSE;
	xTmpStopCycle:=FALSE;
	xStartMainPrc:=FALSE;
	xTmpStop:=FALSE;
	xInitMainCtr:=FALSE;
	xStartMainCtr:=FALSE;
	xStart:=FALSE;
	xSetError:=FALSE;
	xQuitErr:=FALSE;
	xError:=FALSE;
	diErrorNr:=0;
	xInitError:=FALSE;
	xFreeze:=FALSE;
	xAbord:=FALSE;
	xTmpAbord:=FALSE;
	xSetEndPrc:=FALSE;
	xStartProcess:=FALSE;
(*08.07.2014: KFS	{	*)
	xWarmUp:= xWarmUpCycle:= FALSE;
	xWarmUpDone:=FALSE;
(*08.07.2014: KFS	}	*)
	T_ExchgParam.T_StationCommon.T_AutoGeometryPara.xMoveTableStuderBW := FALSE; (*SOA*)
END_IF;
END_FUNCTION_BLOCK

(* POU GENERAL/FB_CheckToolGeometryPara, ST *)
FUNCTION_BLOCK FB_CheckToolGeometryPara
VAR_INPUT
	iProcessNr:INT;	(* 1=AutoGeometry, 2=AutoGroove *)
	T_GeometryCommon:ST_GEOMETRY_COMMON;
	T_AutoGeometryPara:ST_EXCHG_PARAM_AUTOGEOMETRY;
	T_AutoGroovePara:ST_EXCHG_PARAM_AUTOGROOVE;
	T_ProcessPara:ST_EXCHG_PARAM_PROCESS;
	rToolDiameter:REAL;
(*22.12.2009: KFS 	{    *)
	xMicroRodActive: BOOL;				(* choice of the machine MicroWire or MicroRod *)
(*04.04.2011: KFS	{
	rOffsetMaxToolLength:REAL;
04.04.2011: KFS	}   *)
(*22.12.2009: KFS 	}   *)
END_VAR
VAR_OUTPUT
	xError:BOOL;		(* errorflag *)
	diErrorNr: DINT;	(* number of the caused error *)
(*22.12.2009: KFS 	{    *)
	xMultiCycleGrindFeedGeometry: BOOL;				(* choice of multicycle for MicroRod *)
(*22.12.2009: KFS 	}   *)
END_VAR
VAR
	ii: INT;
	rToolLength: REAL;
	rToolDiamterMax: REAL;
	rToolDiamterMin: REAL;
END_VAR
(****************************************************************************************************************************************************)
(***********                         check the settled value of the geometry and set an error if the value is not correct                         ************)
(****************************************************************************************************************************************************)
(* Check ToolLength *)
	rToolLength:=0;
	diErrorNr:=0;
	xError:=FALSE;
	xMultiCycleGrindFeedGeometry:= FALSE;
	FOR ii:=1 TO 6 DO
		IF T_GeometryCommon.T_Geometry.axActiveSection[ii] THEN
			rToolLength:=rToolLength + T_GeometryCommon.T_Geometry.arSectionLength[ii];
		END_IF;
	END_FOR;
(*
	IF (iProcessNr = 1) THEN
		IF T_AutoGeometryPara.xPlungeActivationGeometry THEN
			rToolLength:=rToolLength + (T_AutoGeometryPara.rPlungeLengthToolFeedGeometry / 10.0);
		END_IF;
		IF T_AutoGeometryPara.xDisplaceActivationGeometry THEN
			rToolLength:=rToolLength + (T_AutoGeometryPara.rDisplaceLengthToolFeedGeometry / 10.0);
		END_IF;
		IF (T_AutoGeometryPara.iCycleGeometry > 1) THEN
			rToolLength:=rToolLength * INT_TO_REAL(T_AutoGeometryPara.iCycleGeometry);
		END_IF;
	END_IF;
	IF (iProcessNr = 2) THEN
		IF T_AutoGroovePara.xPlungeActivationGroove THEN
			rToolLength:=rToolLength + (T_AutoGroovePara.rPlungeLengthToolFeedGroove / 10.0);
		END_IF;
		IF T_AutoGroovePara.xDisplaceActivationGroove THEN
			rToolLength:=rToolLength + (T_AutoGroovePara.rDisplaceLengthToolFeedGroove / 10.0);
		END_IF;
	END_IF;
*)
	(*22.12.2009: KFS 	{    *)
	IF xMicroRodActive THEN
		IF rToolLength > (T_GeometryCommon.rMaxToolLength - T_ProcessPara.rStartPosToolFeedAuto * 0.1(* - rOffsetMaxToolLength*) ) THEN
			diErrorNr:=16#F201;	(* Settled parameter for ToolLength is to long *)
		END_IF;
		IF rToolLength < T_GeometryCommon.rMinToolLength THEN
			diErrorNr:=16#F202;	(* Settled parameter for ToolLength is to short *)
		END_IF;
	ELSE
		IF rToolLength > T_GeometryCommon.rMaxToolLength THEN
			diErrorNr:=16#F201;	(* Settled parameter for ToolLength is to long *)
		END_IF;
		IF rToolLength < T_GeometryCommon.rMinToolLength THEN
			diErrorNr:=16#F202;	(* Settled parameter for ToolLength is to short *)
		END_IF;
	END_IF;

	(*22.12.2009: KFS	}   *)
	(*09.12.2022: SOA	{   *)
(* Check ToolDiamter in case of the prisma *)
	rToolDiamterMax:=0;
	FOR ii:=1 TO 6 DO
		IF T_GeometryCommon.T_Geometry.axActiveSection[ii] THEN
			IF (T_GeometryCommon.T_Geometry.arStartDiameter[ii] > rToolDiamterMax) THEN
				rToolDiamterMax:=T_GeometryCommon.T_Geometry.arStartDiameter[ii];
			END_IF;
			IF (T_GeometryCommon.T_Geometry.arEndDiameter[ii] > rToolDiamterMax) THEN
				rToolDiamterMax:=T_GeometryCommon.T_Geometry.arEndDiameter[ii];
			END_IF;
		END_IF;
	END_FOR;
	rToolDiamterMin:=999999;
	FOR ii:=1 TO 6 DO
		IF T_GeometryCommon.T_Geometry.axActiveSection[ii] THEN
			IF (T_GeometryCommon.T_Geometry.arStartDiameter[ii] < rToolDiamterMin) THEN
				rToolDiamterMin:=T_GeometryCommon.T_Geometry.arStartDiameter[ii];
			END_IF;
			IF (T_GeometryCommon.T_Geometry.arEndDiameter[ii] < rToolDiamterMin) THEN
				rToolDiamterMin:=T_GeometryCommon.T_Geometry.arEndDiameter[ii];
			END_IF;
		END_IF;
	END_FOR;
	IF (rToolDiamterMax > T_GeometryCommon.rMaxToolDiameter) THEN
		diErrorNr:=16#F203;	(* Settled parameter for ToolDiameter is to big *)
	END_IF;
	IF (rToolDiamterMin < T_GeometryCommon.rMinToolDiameter) THEN
		diErrorNr:=16#F204;	(* Settled parameter for ToolDiameter is to small *)
	END_IF;
	(*22.12.2009: KFS 	{    *)
(* Check activation for multicycle of the AutoGeometry *)
	IF xMicroRodActive THEN
		IF ( (rToolDiameter - rToolDiamterMin) > T_AutoGeometryPara.rPlungeCycleGrindFeedGeometry ) THEN
			xMultiCycleGrindFeedGeometry := TRUE;
		END_IF;
	END_IF;
	(*22.12.2009: KFS 	}    *)
(* Check the passage from one section to another section if equal *)
	FOR ii:=1 TO 6 DO
		IF T_GeometryCommon.T_Geometry.axActiveSection[ii] THEN
			IF (ii < 6) THEN
				IF T_GeometryCommon.T_Geometry.axActiveSection[ii+ 1] THEN
					IF (T_GeometryCommon.T_Geometry.arEndDiameter[ii] <> T_GeometryCommon.T_Geometry.arStartDiameter[ii + 1]) THEN
						diErrorNr:=16#F205;	(* At least a passage of a section is not equal *)
					END_IF;
				END_IF;
			END_IF;
		END_IF;
	END_FOR;
(* Check ToolDiamter in case of the settled ToolDiameter *)
	rToolDiamterMax:=0;
	FOR ii:=1 TO 6 DO
		IF T_GeometryCommon.T_Geometry.axActiveSection[ii] THEN
			IF (T_GeometryCommon.T_Geometry.arStartDiameter[ii] > rToolDiamterMax) THEN
				rToolDiamterMax:=T_GeometryCommon.T_Geometry.arStartDiameter[ii];
			END_IF;
			IF (T_GeometryCommon.T_Geometry.arEndDiameter[ii] > rToolDiamterMax) THEN
				rToolDiamterMax:=T_GeometryCommon.T_Geometry.arEndDiameter[ii];
			END_IF;
		END_IF;
	END_FOR;
	IF (rToolDiamterMax > rToolDiameter) THEN
		diErrorNr:=16#F206;	(* At least one settled diameter is bigger than the ToolDiameter *)
	END_IF;
	IF (diErrorNr <> 0) THEN
		xError:=TRUE;
	END_IF;
(*09.12.2022: SOA	}	 *)
END_FUNCTION_BLOCK

(* POU PRG_PROCESS_LAYER4/FB_PROCESS/FB_PrcAutoGroove, ST *)
FUNCTION_BLOCK FB_PrcAutoGroove
VAR_INPUT
	xMicroRodActive: BOOL;				(* choice of the machine MicroWire or MicroRod *)
	xBeckhoffDriveActive: BOOL;			(* choice of the axis Beckhoff or EcoStep *)
	T_NovRAMData:ST_DATA_RETAIN;	(* Novram structure for all Machine parameter *)
END_VAR
VAR_IN_OUT
	xStart : BOOL;							(* start a process *)
	xStop : BOOL;							(* stop a process *)
	xQuitErr : BOOL;						(* quit an error *)
	xAbord : BOOL;						(* abord a process *)
	T_Station : ST_STATION;				(* data structure of the stationlevel *)
	T_Process : ST_PROCESS;			(* data strucuture of the processlevel *)
	xReset : BOOL;						(* reset the FB *)
	T_ExchgParam:ST_QVIS_EXCHG_PARAM;	(* data structure of the visualisation *)
	xDoNotMoveGrindPosition:BOOL;		(* choice of the AutoGroove process, TRUE=override the GrindAxis position with the ToolDiameter, FALSE=no overriding *)
	xPlungeActive:BOOL;					(* TRUE=Plunge on AutoGroove active, FALSE=Plunge on AutoGroove deactivatet *)
END_VAR
VAR_OUTPUT
	xEnd : BOOL;							(* Endflag of the process *)
	xError : BOOL;							(* Errorflag of the process *)
	diErrorNr : DINT;						(* Error number of the process *)
END_VAR
VAR
	iStepPrc: INT;
	xInitStep: BOOL;
	xSetError: BOOL;
	xSetEnd: BOOL;
	xStartMainCtr: BOOL;
	xStartMainPrc: BOOL;
	xInitMainCtr: BOOL;
	xFreeze: BOOL;
	xInitError: BOOL;
	iStepError: INT;
	xTmpStop: BOOL;
	xSetTmpError: BOOL;
	xTmpAbord: BOOL;
	diTmpErrNr: DINT;
	xSetEndPrc : BOOL;
	iTmpFunctionNr:INT;
	xStopFctStation1: BOOL;
	iStepStop: INT;
	FBCheckToolGeometryPara: FB_CheckToolGeometryPara;
	iTmpStationFunctionNr: INT;
	xStartProcess: BOOL;
	TONStartTimer: TON;
	tStepTime: TIME;
	TONStartTimer1: TON;
	rCheckStartPosition: REAL;
	(*22.12.2009: KFS	{ *)
	iNumberOfGrooves: INT;
	lrAxisToolLeftActuelPosition: LREAL;
	rStartPosAutoGrooveToolRotation: LREAL;
	rOffsetStartPositionGrooves: REAL;
	xOneTimeCheckGeometry:BOOL;
	(*22.12.2009: KFS	} *)
	rMaxTol: REAL:= 5.0;
	xNotFirstGrooveCycle: BOOL;
	TONStartTimer2: TON; (*SOA*)
END_VAR
(****************************************************************************************************************************************************)
(***********                                      This Functionblock define the process for the AutoGroove                                                         ************)
(****************************************************************************************************************************************************)

(******************************************************************************************************************************************)
(****************************				           Reset Function Part                                                 *****************************)
(******************************************************************************************************************************************)
IF xReset THEN
	xReset:=FALSE;
	xSetEnd:=TRUE;
END_IF;
(******************************************************************************************************************************************)
(****************************				              Error Controlling Part                                            *****************************)
(******************************************************************************************************************************************)
IF (xSetError OR T_Station.TControl.xError) AND NOT(xSetEnd) THEN
	IF NOT(xInitError) THEN
		iStepError:=100;
		xInitError:=TRUE;
		IF NOT(xSetError) THEN
			xSetError:=TRUE;
			xSetTmpError:=FALSE;
		ELSE
			xSetTmpError:=TRUE;
		END_IF;
	END_IF;
	CASE iStepError OF
		100:	IF T_Station.TControl.xError THEN
				diErrorNr:=T_Station.TControl.diErrorNr;
			END_IF;
			IF xSetTmpError THEN
				diErrorNr:=diTmpErrNr;
			END_IF;
			iStepError:=200;
		200:	IF xSetTmpError THEN
				xSetTmpError:=FALSE;
				xStopFctStation1:=FALSE;
				iStepError:=300;
			ELSE
				IF NOT(T_Station.TControl.xError) AND NOT(T_Station.TControl.xEnd) THEN
					IF (T_Station.TControl.iFunctNr = 1) THEN
						T_Station.TControl.xStop:=TRUE;
						xStopFctStation1:=TRUE;
					ELSE
						xStopFctStation1:=FALSE;
					END_IF;
				END_IF;
				iStepError:=300;
			END_IF;
		300:	IF xStopFctStation1 THEN
				IF NOT(T_Station.TControl.xStop) THEN
					xStopFctStation1:=FALSE;
				END_IF;
			END_IF;
			IF NOT(xStopFctStation1) THEN
				xError:=TRUE;
				iStepError:=400;
			END_IF;
		400:	IF xQuitErr THEN
				T_Station.TControl.xQuitError:=T_Station.TControl.xError;
				iStepError:=500;
			END_IF;
		500: IF NOT(T_Station.TControl.xQuitError) THEN
				xSetEnd:=TRUE;
			END_IF;
	END_CASE;
END_IF;
(******************************************************************************************************************************************)
(****************************				              Main Controlling Part                                            *****************************)
(******************************************************************************************************************************************)
IF (xStart OR xStartMainCtr) AND NOT(xSetEnd) AND NOT(xSetError) THEN
	IF NOT (xInitMainCtr) THEN
		iStepPrc:=10;
		xInitMainCtr:=TRUE;
		xStartMainCtr:=TRUE;
		xStart:=FALSE;
		xEnd:=FALSE;
		xSetEndPrc:=FALSE;
		iTmpFunctionNr:=1;
		xAbord:=FALSE;
		T_ExchgParam.T_InfoValueCommon.rActualWireFeedPosition:=0.0;
		T_ExchgParam.T_InfoValueCommon.rActualWireFeedSpeed:=0.0;
		(*22.12.2009: KFS 	{ *)
		T_Station.rStartPosAutoGrooveToolRotation:=0.0;
		rStartPosAutoGrooveToolRotation:=0.0;
		lrAxisToolLeftActuelPosition:=0.0;
		(*22.12.2009: KFS 	} *)
	END_IF;
	IF xStop AND NOT(xTmpStop) THEN
		xTmpStop:=TRUE;
		iStepStop:=1;
	END_IF;
	IF xTmpStop THEN
		CASE iStepStop OF
		1:	IF NOT(T_Station.TControl.xEnd) THEN
				T_Station.TControl.xStop:=TRUE;
				iStepStop:=10;
			ELSE
				iStepStop:=20;
			END_IF;
		10:	IF NOT(T_Station.TControl.xStop) THEN
				iStepStop:=20;
			END_IF;
		20:	IF NOT(T_Station.TControl.xStart) AND T_Station.TControl.xEnd THEN
				T_Station.TControl.iFunctNr:=4;
				T_Station.TControl.xStart:=TRUE;
				T_Station.THardware.TAxisGrindFeeder.T_CtrleSingle.lrAcceleration:=T_NovRAMData.T_Standard.T_TeachINGrindFeeder.rAcceleration;
				T_Station.THardware.TAxisGrindFeeder.T_CtrleSingle.lrDecceleration:=T_NovRAMData.T_Standard.T_TeachINGrindFeeder.rDeceleration;
				T_Station.THardware.TAxisGrindFeeder.T_CtrleSingle.lrPosition:=	T_NovRAMData.T_ProcessImageData.T_ProcessPara.rToolDiameterProcess +
																			T_NovRAMData.T_ProcessImageData.T_ProcessPara.rSecurityPosGrindFeedProcess;
				T_Station.THardware.TAxisGrindFeeder.T_CtrleSingle.lrVelocity:=T_NovRAMData.T_ProcessImageData.T_ProcessPara.rSpeedBackwardGrindFeed;
				iStepStop:=30;
			END_IF;
		(* Check Active Movement of the Axis *)
		30:	IF NOT(T_Station.TControl.xStart) AND T_Station.TControl.xEnd THEN
				T_Station.TControl.iFunctNr:=18;	(* Check Axis Movement, and stop it if moves *)
				T_Station.TControl.xStart:=TRUE;
				iStepStop:=40;
			END_IF;
		40:	IF NOT(T_Station.TControl.xStart) AND T_Station.TControl.xEnd THEN
				xStartMainPrc:=FALSE;
				xInitStep:=FALSE;
				iStepPrc:=0;
				xSetEnd:=TRUE;
				RETURN;
			END_IF;
		END_CASE;
		RETURN;
	END_IF;
	IF NOT(xStartMainPrc) THEN
		xStartMainPrc:=TRUE;
	END_IF;
END_IF;
(******************************************************************************************************************************************)
(****************************		               Controlling of the ToolLeft Position                                   *****************************)
(******************************************************************************************************************************************)
IF  T_Station.THardware.TAxisToolLeft.T_LiveValue.lrActualPositionRelativ <> 0THEN
	IF xMicroRodActive THEN
		lrAxisToolLeftActuelPosition:=T_Station.THardware.TAxisToolLeft.T_LiveValue.lrActualPositionRelativ;
	END_IF;
END_IF;
(******************************************************************************************************************************************)
(****************************				             Main Procedure Part                                             *****************************)
(******************************************************************************************************************************************)
IF xStartProcess THEN
	TONStartTimer(IN:=TRUE,PT:=T#1s);
	IF TONStartTimer.Q THEN
		TONStartTimer(IN:=FALSE);
		IF (T_ExchgParam.T_InfoValueCommon.tAutoTimeLeft >= T#1s) THEN
			T_ExchgParam.T_InfoValueCommon.tAutoTimeLeft:=T_ExchgParam.T_InfoValueCommon.tAutoTimeLeft - T#1s;
		ELSE
			T_ExchgParam.T_InfoValueCommon.tAutoTimeLeft:=T#0s;
		END_IF;
	END_IF;
	tStepTime:=T_ExchgParam.T_InfoValueCommon.tAutoTimeTotal / 100;
	TONStartTimer1(IN:=TRUE,PT:=tStepTime);
	IF TONStartTimer1.Q THEN
		TONStartTimer1(IN:=FALSE);
		T_ExchgParam.T_InfoValueCommon.bProgressbarAutoGroove:=T_ExchgParam.T_InfoValueCommon.bProgressbarAutoGroove + 1;
		IF (T_ExchgParam.T_InfoValueCommon.bProgressbarAutoGroove >= 100) THEN
			T_ExchgParam.T_InfoValueCommon.bProgressbarAutoGroove:=100;
		END_IF;
	END_IF;
ELSE
	TONStartTimer(IN:=FALSE);
	TONStartTimer1(IN:=FALSE);
END_IF;
IF xStartMainPrc AND NOT(xSetEnd) AND NOT(xSetError) THEN
	CASE iStepPrc OF
		(* Check first if the AutoGroove is available to start it *)
		10:	T_ExchgParam.T_InfoValueCommon.iCountDownGrooveCycle:=1;
			T_Station.THardware.TAxisToolLeft.T_CtrleSingle.lrAcceleration:=T_NovRAMData.T_Standard.T_TeachINToolLeft.rAcceleration;
			T_Station.THardware.TAxisToolLeft.T_CtrleSingle.lrDecceleration:=T_NovRAMData.T_Standard.T_TeachINToolLeft.rDeceleration;
			T_Station.THardware.TAxisToolCenter.T_CtrleSingle.lrAcceleration:=T_NovRAMData.T_Standard.T_TeachINToolCenter.rAcceleration;
			T_Station.THardware.TAxisToolCenter.T_CtrleSingle.lrDecceleration:=T_NovRAMData.T_Standard.T_TeachINToolCenter.rDeceleration;
			T_Station.THardware.TAxisToolRight.T_CtrleSingle.lrAcceleration:=T_NovRAMData.T_Standard.T_TeachINToolRight.rAcceleration;
			T_Station.THardware.TAxisToolRight.T_CtrleSingle.lrDecceleration:=T_NovRAMData.T_Standard.T_TeachINToolRight.rDeceleration;
			T_Station.THardware.TAxisToolFeeder.T_CtrleSingle.lrAcceleration:=T_NovRAMData.T_Standard.T_TeachINToolFeeder.rAcceleration;
			T_Station.THardware.TAxisToolFeeder.T_CtrleSingle.lrDecceleration:=T_NovRAMData.T_Standard.T_TeachINToolFeeder.rDeceleration;
			T_Station.THardware.TAxisGrindFeeder.T_CtrleSingle.lrAcceleration:=T_NovRAMData.T_Standard.T_TeachINGrindFeeder.rAcceleration;
			T_Station.THardware.TAxisGrindFeeder.T_CtrleSingle.lrDecceleration:=T_NovRAMData.T_Standard.T_TeachINGrindFeeder.rDeceleration;
			(* Only for MicroRod, check if the tool is clamped *)
			IF xMicroRodActive THEN
				(*22.12.2009: KFS	{ *)
				(*Added control if all cylinder for the tool are activated*)
				IF T_Station.THardware.TCylToolTension.T_CtrleCyl.xStatePosOn OR
				     T_Station.THardware.TCylToolLeftActive.T_CtrleCyl.T_Standard.xActivOn OR
 				     T_Station.THardware.TCylToolRightActive.T_CtrleCyl.T_Standard.xActivOn  OR
				   (* T_Station.THardware.TCylToolCenterActive.T_CtrleCyl.T_Standard.xActivOn OR*)	(* IGS auskommentiert, diesen Zyl gibts auf der M3 nicht *)
				     NOT(T_Station.THardware.TCylToolPrismaLeftActive.T_CtrleCyl.T_Standard.xActivOn) OR
				     NOT(T_Station.THardware.TCylToolPrismaRightActive.T_CtrleCyl.T_Standard.xActivOn) 	THEN
					xSetError:=TRUE;
					diTmpErrNr:=2;			(* Tool is not clamped *)
				END_IF;
				(*22.12.2009: KFS	} *)
			END_IF;
			(* Only for MicroRod, check if the Machine is referenced *)
			IF xMicroRodActive THEN
				IF NOT(T_Station.TControl.xReferenced) THEN
					xSetError:=TRUE;
					diTmpErrNr:=1;	(* Machine is not referenced *)
					RETURN;
				END_IF;
			END_IF;
			(* Only for MicroRod, check if the second procedure of AutoGroove is active if the ToolFeeder is on the StartPos *)
			IF xMicroRodActive THEN
				IF xDoNotMoveGrindPosition THEN
					IF xPlungeActive THEN
						(* less than 1mm is alowed of the position of the ToolFeeder from the StartPosition + the ToolFeed lenght by activated Plunge *)
						rCheckStartPosition:=	ABS((T_NovRAMData.T_ProcessImageData.T_ProcessPara.rStartPosToolFeedAuto +
												T_NovRAMData.T_ProcessImageData.T_AutoGroovePara.rPlungeLengthToolFeedGroove) -
												T_Station.THardware.TAxisToolFeeder.T_LiveValue.lrActualPosition);
						IF (rCheckStartPosition > 1.0) THEN
							xSetError:=TRUE;
							diTmpErrNr:=4;	(* ToolFeeeder is not on the StartPosition *)
							RETURN;
						END_IF;
					ELSE
						(* less than 1mm is alowed of the position of the ToolFeeder from the StartPosition *)
						IF (ABS(T_NovRAMData.T_ProcessImageData.T_ProcessPara.rStartPosToolFeedAuto - T_Station.THardware.TAxisToolFeeder.T_LiveValue.lrActualPosition) > 1.0) THEN
							xSetError:=TRUE;
							diTmpErrNr:=4;	(* ToolFeeeder is not on the StartPosition *)
							RETURN;
						END_IF;
					END_IF;
				END_IF;
			END_IF;
			(*22.12.2009: KFS	{ *)
			(* Only for MicroRod, set number of grooves and StartPosAutoGrooveToolRotation *)
			IF xMicroRodActive THEN
				iNumberOfGrooves:= T_NovRAMData.T_ProcessImageData.T_AutoGroovePara.iNumberOfGrooves;
				xNotFirstGrooveCycle:=FALSE;
				IF T_NovRAMData.T_ProcessImageData.T_AutoGroovePara.iNumberOfGrooves >0 THEN
					rOffsetStartPositionGrooves:= 360.0 / T_NovRAMData.T_ProcessImageData.T_AutoGroovePara.iNumberOfGrooves;
				END_IF;
			END_IF;
			(*22.12.2009: KFS	}*)
			xStartMainPrc:=FALSE;
			xInitStep:=FALSE;
			iStepPrc:=11;
		(* Set the ToolTension force *)
		11:	IF NOT(xInitStep) THEN
				xInitStep:=TRUE;
				T_Station.THardware.TCylToolTension.T_CtrleCyl.iFunction:=2;	(* activate the ToolTension *)
				T_Station.THardware.TCylToolTension.T_CtrleCyl.T_AnalogCylinder.rForceIn:=T_NovRAMData.T_ProcessImageData.T_ProcessPara.rToolTensionProcess;
				IF xMicroRodActive THEN
					T_Station.THardware.TCylToolTension.T_Config.tDelayOn:=T#1s;
				ELSE
					T_Station.THardware.TCylToolTension.T_Config.tDelayOn:=T#0s;
				END_IF;
				T_Station.THardware.TCylToolTension.T_CtrleCyl.xExecute:=TRUE;
			END_IF;
			IF NOT(T_Station.THardware.TCylToolTension.T_CtrleCyl.xExecute) AND T_Station.THardware.TCylToolTension.T_CtrleCyl.xDone THEN
				(* Only for MicroRod, check if the tool is clamped *)
				IF xMicroRodActive THEN
					IF T_Station.THardware.TCylToolTension.T_CtrleCyl.xStatePosOn THEN
						xSetError:=TRUE;
						diTmpErrNr:=2;			(* Tool is not clamped *)
						RETURN;
					END_IF;
				END_IF;
				iStepPrc:=20;
				xStartMainPrc:=FALSE;
				xInitStep:=FALSE;
			END_IF;
		(* Switch First all Axis the power supply on *)
		20:	IF NOT(xInitStep) THEN
				xInitStep:=TRUE;
				T_Station.TControl.iFunctNr:=16;
				T_Station.TControl.xStart:=TRUE;
			END_IF;
			IF NOT(T_Station.TControl.xStart) AND T_Station.TControl.xEnd THEN
				iStepPrc:=30;
				xStartMainPrc:=FALSE;
				xInitStep:=FALSE;
				iTmpStationFunctionNr:=6;
				T_Station.THardware.TAxisToolLeft.T_CtrleSingle.rSetPosition:=0.0;
				T_Station.THardware.TAxisToolCenter.T_CtrleSingle.rSetPosition:=0.0;
				T_Station.THardware.TAxisToolRight.T_CtrleSingle.rSetPosition:=0.0;
				T_Station.THardware.TAxisToolFeeder.T_CtrleSingle.rSetPosition:=0.0;
			END_IF;
		(* Reset the Position of the Axis *)
		30:	IF NOT(xInitStep) THEN
				xInitStep:=TRUE;
				(* 6=ToolLeft, 7=ToolCenter, 8=ToolRight, 9=ToolFeeder *)
				T_Station.TControl.iFunctNr:=iTmpStationFunctionNr;
				T_Station.TControl.xStart:=TRUE;
			END_IF;
			IF NOT(T_Station.TControl.xStart) AND T_Station.TControl.xEnd THEN
				iTmpStationFunctionNr:=iTmpStationFunctionNr + 1;
				IF NOT(xMicroRodActive) AND (iTmpStationFunctionNr = 7) THEN
					iTmpStationFunctionNr:=iTmpStationFunctionNr + 1;
				END_IF;
				IF xMicroRodActive AND (iTmpStationFunctionNr = 9) THEN
					iTmpStationFunctionNr:=iTmpStationFunctionNr + 1;
				END_IF;
				xStartMainPrc:=FALSE;
				xInitStep:=FALSE;
				IF (iTmpStationFunctionNr < 10) THEN
					iStepPrc:=30;
				ELSE
					IF NOT(xDoNotMoveGrindPosition) THEN
						iStepPrc:=40;
					ELSE
						iStepPrc:=70;	(* Start with the working without to adjust the GrindFeeder on the Position of the ToolDiameter *)
					END_IF;
					(*10.09.2010: KFS   { Save StartPos of ToolRotation*)
					rStartPosAutoGrooveToolRotation:=T_Station.THardware.TAxisToolLeft.T_LiveValue.lrActualPositionRelativ;
					(*10.09.2010: KFS	} *)
				END_IF;
			END_IF;
		(* GrindFeeder Set Absolut to Security Position *)
		40:	IF NOT(xInitStep) THEN
				xInitStep:=TRUE;
				T_Station.TControl.iFunctNr:=4;
				T_Station.TControl.xStart:=TRUE;
				T_Station.THardware.TAxisGrindFeeder.T_CtrleSingle.lrAcceleration:=T_NovRAMData.T_Standard.T_TeachINGrindFeeder.rAcceleration;
				T_Station.THardware.TAxisGrindFeeder.T_CtrleSingle.lrDecceleration:=T_NovRAMData.T_Standard.T_TeachINGrindFeeder.rDeceleration;
				T_Station.THardware.TAxisGrindFeeder.T_CtrleSingle.lrPosition:=	T_NovRAMData.T_ProcessImageData.T_ProcessPara.rToolDiameterProcess +
																			T_NovRAMData.T_ProcessImageData.T_ProcessPara.rSecurityPosGrindFeedProcess;
				T_Station.THardware.TAxisGrindFeeder.T_CtrleSingle.lrVelocity:=T_NovRAMData.T_ProcessImageData.T_ProcessPara.rSpeedBackwardGrindFeed;
			END_IF;
			IF NOT(T_Station.TControl.xStart) AND T_Station.TControl.xEnd THEN
				IF xMicroRodActive THEN
					iStepPrc:=50;
				ELSE
					iStepPrc:=60;
				END_IF;
				xStartMainPrc:=FALSE;
				xInitStep:=FALSE;
			END_IF;
		(* Only for MicroRod-->Set ToolFeed Absolut to the Zero Position*)
		50:	IF NOT(xInitStep) THEN
(* 04.04.2011: KFS	{ 	Neu wird die Längeneinstellung des ToolFeeders nicht mehr kontrolliert und direkt auf die StartPos gefahren(vormals RefPos)!
				xInitStep:=TRUE;
				T_Station.TControl.iFunctNr:=14;
				T_Station.TControl.xStart:=TRUE;
				T_Station.THardware.TAxisToolFeeder.T_CtrleSingle.lrAcceleration:=T_NovRAMData.T_Standard.T_TeachINToolFeeder.rAcceleration;
				T_Station.THardware.TAxisToolFeeder.T_CtrleSingle.lrDecceleration:=T_NovRAMData.T_Standard.T_TeachINToolFeeder.rDeceleration;
				T_Station.THardware.TAxisToolFeeder.T_CtrleSingle.lrPosition:=0.0;
				T_Station.THardware.TAxisToolFeeder.T_CtrleSingle.lrVelocity:=T_NovRAMData.T_ProcessImageData.T_ProcessPara.rSpeedStartPosToolFeedProcess;
			END_IF;
			IF NOT(T_Station.TControl.xStart) AND T_Station.TControl.xEnd THEN
 04.04.2011: KFS	}	*)
				FBCheckToolGeometryPara(	iProcessNr:= 1,
											T_GeometryCommon:= T_ExchgParam.T_GeometryCommon,
											T_AutoGeometryPara:= T_NovRAMData.T_ProcessImageData.T_AutoGeometryPara,
											T_AutoGroovePara:= T_NovRAMData.T_ProcessImageData.T_AutoGroovePara,
											T_ProcessPara:= T_NovRamData.T_ProcessImageData.T_ProcessPara,
											rToolDiameter:=T_NovRAMData.T_ProcessImageData.T_ProcessPara.rToolDiameterProcess,
											xMicroRodActive:= xMicroRodActive,
											(*rOffsetMaxToolLength:= T_Station.THardware.TToolFeederWorkLength.T_CtrleCyl.T_Analog.rLengthIn*));
				IF FBCheckToolGeometryPara.xError THEN
					xSetError:=TRUE;
					diTmpErrNr:=FBCheckToolGeometryPara.diErrorNr;
					RETURN;
				END_IF;
				iStepPrc:=55;
				xStartMainPrc:=FALSE;
				xInitStep:=FALSE;
			END_IF;
		(* Only for MicroRod-->Set ToolFeed Absolut to the StartPosition *)
		55:	IF NOT(xInitStep) THEN
				xInitStep:=TRUE;
				T_Station.TControl.iFunctNr:=14;
				T_Station.TControl.xStart:=TRUE;
				T_Station.THardware.TAxisToolFeeder.T_CtrleSingle.lrAcceleration:=T_NovRAMData.T_Standard.T_TeachINToolFeeder.rAcceleration;
				T_Station.THardware.TAxisToolFeeder.T_CtrleSingle.lrDecceleration:=T_NovRAMData.T_Standard.T_TeachINToolFeeder.rDeceleration;
				T_Station.THardware.TAxisToolFeeder.T_CtrleSingle.lrPosition:=T_NovRAMData.T_ProcessImageData.T_ProcessPara.rStartPosToolFeedAuto;
				T_Station.THardware.TAxisToolFeeder.T_CtrleSingle.lrVelocity:=T_NovRAMData.T_ProcessImageData.T_ProcessPara.rSpeedStartPosToolFeedProcess;
			END_IF;
			IF NOT(T_Station.TControl.xStart) AND T_Station.TControl.xEnd THEN
				iStepPrc:=60;
				xStartMainPrc:=FALSE;
				xInitStep:=FALSE;
			END_IF;
		(* GrindFeeder Set Absolut to ToolDiameter minus the offset with the fast speed *)
		60:	IF NOT(xInitStep) THEN
				xInitStep:=TRUE;
				T_Station.TControl.iFunctNr:=4;
				T_Station.TControl.xStart:=TRUE;
				T_Station.THardware.TAxisGrindFeeder.T_CtrleSingle.lrAcceleration:=T_NovRAMData.T_Standard.T_TeachINGrindFeeder.rAcceleration;
				T_Station.THardware.TAxisGrindFeeder.T_CtrleSingle.lrDecceleration:=T_NovRAMData.T_Standard.T_TeachINGrindFeeder.rDeceleration;
				T_Station.THardware.TAxisGrindFeeder.T_CtrleSingle.lrPosition:=T_NovRAMData.T_ProcessImageData.T_ProcessPara.rToolDiameterProcess + T_NovRAMData.T_ProcessImageData.T_ProcessPara.rOffsetBeforeToolDiaGrindFeedProcess;
				T_Station.THardware.TAxisGrindFeeder.T_CtrleSingle.lrVelocity:=T_NovRAMData.T_ProcessImageData.T_ProcessPara.rSpeedForwardFastGrindFeed;
			END_IF;
			IF NOT(T_Station.TControl.xStart) AND T_Station.TControl.xEnd THEN
				xStartMainPrc:=FALSE;
				xInitStep:=FALSE;
				iStepPrc:=70;
			END_IF;
		(* Working AutoGroove *)
		70:	IF NOT(xInitStep) THEN
				xStartProcess:=TRUE;
				xInitStep:=TRUE;
				T_Station.TControl.iFunctNr:=12;
				T_Station.TControl.xStart:=TRUE;
				IF xNotFirstGrooveCycle THEN
					T_ExchgParam.T_InfoValueCommon.iCountDownGrooveCycle:=T_ExchgParam.T_InfoValueCommon.iCountDownGrooveCycle +1;
				ELSE
					xNotFirstGrooveCycle:= TRUE;
				END_IF;
			END_IF;
			IF NOT(T_Station.TControl.xStart) AND T_Station.TControl.xEnd THEN
				xStartMainPrc:=FALSE;
				xInitStep:=FALSE;
				iStepPrc:=80;
				RETURN;
			END_IF;
			(* Only for MicroRod, check if the tool is clamped *)
			IF xMicroRodActive THEN
				IF T_Station.THardware.TCylToolTension.T_CtrleCyl.xStatePosOn THEN
					xStartMainPrc:=FALSE;
					xInitStep:=FALSE;
					iStepPrc:=71;
					RETURN;
				END_IF;
			END_IF;
		(* Stop the Process, because the Tool is broken *)
		71:	IF NOT(xInitStep) THEN
				xInitStep:=TRUE;
				T_Station.TControl.xStop:=TRUE;
			END_IF;
			IF NOT(T_Station.TControl.xStart) AND T_Station.TControl.xEnd THEN
				xStartMainPrc:=FALSE;
				xInitStep:=FALSE;
				iStepPrc:=72;
			END_IF;
		(* Set the GrindFeeder to the security Position *)
		72:	IF NOT(xInitStep) THEN
				xInitStep:=TRUE;
				T_Station.TControl.iFunctNr:=4;
				T_Station.TControl.xStart:=TRUE;
				T_Station.THardware.TAxisGrindFeeder.T_CtrleSingle.lrAcceleration:=T_NovRAMData.T_Standard.T_TeachINGrindFeeder.rAcceleration;
				T_Station.THardware.TAxisGrindFeeder.T_CtrleSingle.lrDecceleration:=T_NovRAMData.T_Standard.T_TeachINGrindFeeder.rDeceleration;
				T_Station.THardware.TAxisGrindFeeder.T_CtrleSingle.lrPosition:=	T_NovRAMData.T_ProcessImageData.T_ProcessPara.rToolDiameterProcess +
																			T_NovRAMData.T_ProcessImageData.T_ProcessPara.rSecurityPosGrindFeedProcess;
				T_Station.THardware.TAxisGrindFeeder.T_CtrleSingle.lrVelocity:=T_NovRAMData.T_ProcessImageData.T_ProcessPara.rSpeedBackwardGrindFeed;
			END_IF;
			IF NOT(T_Station.TControl.xStart) AND T_Station.TControl.xEnd THEN
				xStartMainPrc:=FALSE;
				xInitStep:=FALSE;
				iStepPrc:=73;
			END_IF;
		(* Check Active Movement of the Axis *)
		73:	IF NOT(xInitStep) THEN
				xInitStep:=TRUE;
				T_Station.TControl.iFunctNr:=18;	(* Check Axis Movement, and stop it if moves *)
				T_Station.TControl.xStart:=TRUE;
			END_IF;
			IF NOT(T_Station.TControl.xStart) AND T_Station.TControl.xEnd THEN
				xSetError:=TRUE;
				diTmpErrNr:=2;			(* Tool is not clamped *)
				RETURN;
			END_IF;
		(* GrindFeeder Set Absolut to Security Position *)
		80:	IF NOT(xInitStep) THEN
				xInitStep:=TRUE;
				T_Station.TControl.iFunctNr:=4;
				T_Station.TControl.xStart:=TRUE;
				T_Station.THardware.TAxisGrindFeeder.T_CtrleSingle.lrAcceleration:=T_NovRAMData.T_Standard.T_TeachINGrindFeeder.rAcceleration;
				T_Station.THardware.TAxisGrindFeeder.T_CtrleSingle.lrDecceleration:=T_NovRAMData.T_Standard.T_TeachINGrindFeeder.rDeceleration;
				T_Station.THardware.TAxisGrindFeeder.T_CtrleSingle.lrPosition:=	T_NovRAMData.T_ProcessImageData.T_ProcessPara.rToolDiameterProcess +
																			T_NovRAMData.T_ProcessImageData.T_ProcessPara.rSecurityPosGrindFeedProcess;
				T_Station.THardware.TAxisGrindFeeder.T_CtrleSingle.lrVelocity:=T_NovRAMData.T_ProcessImageData.T_ProcessPara.rSpeedBackwardGrindFeed;
			END_IF;
			IF NOT(T_Station.TControl.xStart) AND T_Station.TControl.xEnd THEN
				(*10.09.2010: KFS   { Set next  rStartPosAutoGrooveToolRotation*)
				rStartPosAutoGrooveToolRotation:=  LMOD ( (rStartPosAutoGrooveToolRotation + rOffsetStartPositionGrooves) , 360);
				(*10.09.2010: KFS   } *)
				xStartMainPrc:=FALSE;
				xInitStep:=FALSE;
				iStepPrc:=90;
			END_IF;
		(* ToolRotation Stop *)
		90:	IF NOT(xInitStep) THEN
				xInitStep:=TRUE;
				T_Station.TControl.iFunctNr:=3;
				T_Station.TControl.xStart:=TRUE;
				(* ToolLeft --> Master *)
				T_Station.THardware.TAxisToolLeft.T_CtrleSingle.lrAcceleration:=T_NovRAMData.T_Standard.T_TeachINToolLeft.rAcceleration;
				T_Station.THardware.TAxisToolLeft.T_CtrleSingle.lrDecceleration:=T_NovRAMData.T_Standard.T_TeachINToolLeft.rDeceleration;
				IF xMicroRodActive THEN
					(* ToolCenter --> Slave of ToolLeft only by MicroRod *)
					T_Station.THardware.TAxisToolCenter.T_CtrleSingle.lrAcceleration:=T_NovRAMData.T_Standard.T_TeachINToolCenter.rAcceleration;
					T_Station.THardware.TAxisToolCenter.T_CtrleSingle.lrDecceleration:=T_NovRAMData.T_Standard.T_TeachINToolCenter.rDeceleration;
				END_IF;
				(* ToolRight --> Slave of ToolLeft by MicroWire or Slave of ToolRight by MicroRod *)
				T_Station.THardware.TAxisToolRight.T_CtrleSingle.lrAcceleration:=T_NovRAMData.T_Standard.T_TeachINToolRight.rAcceleration;
				T_Station.THardware.TAxisToolRight.T_CtrleSingle.lrDecceleration:=T_NovRAMData.T_Standard.T_TeachINToolRight.rDeceleration;
				IF NOT(xMicroRodActive) THEN
					(* ToolRight --> Slave of ToolRight by MicroWire *)
					T_Station.THardware.TAxisToolFeeder.T_CtrleSingle.lrAcceleration:=T_NovRAMData.T_Standard.T_TeachINToolFeeder.rAcceleration;
					T_Station.THardware.TAxisToolFeeder.T_CtrleSingle.lrDecceleration:=T_NovRAMData.T_Standard.T_TeachINToolFeeder.rDeceleration;
				END_IF;
			END_IF;
			IF NOT(T_Station.TControl.xStart) AND T_Station.TControl.xEnd THEN
				(*10.09.2010: KFS	{ *)
				(*Calculation of the new T_Station.rStartPosAutoGrooveToolRotation*)
				IF xMicroRodActive THEN
					iNumberOfGrooves:=iNumberOfGrooves - 1;
					IF iNumberOfGrooves > 0 THEN
						IF lrAxisToolLeftActuelPosition < rStartPosAutoGrooveToolRotation THEN
							(* Start ToolRotation --> MoveRelativ to rStartPosAutoGrooveToolRotation *)
							T_Station.rStartPosAutoGrooveToolRotation:= rStartPosAutoGrooveToolRotation - lrAxisToolLeftActuelPosition;
						END_IF;
						IF lrAxisToolLeftActuelPosition = rStartPosAutoGrooveToolRotation THEN
							(* Start ToolRotation --> MoveRelativ to rStartPosAutoGrooveToolRotation *)
							T_Station.rStartPosAutoGrooveToolRotation:= 0.0;
						END_IF;
						IF lrAxisToolLeftActuelPosition > rStartPosAutoGrooveToolRotation THEN
							(* Start ToolRotation --> MoveRelativ to rStartPosAutoGrooveToolRotation *)
							T_Station.rStartPosAutoGrooveToolRotation:= 360.0 - ( lrAxisToolLeftActuelPosition - rStartPosAutoGrooveToolRotation);
						END_IF;
						iStepPrc:=55;
					ELSE
		          			iStepPrc:=100;
					END_IF;
				ELSE
					iStepPrc:=100;
				END_IF;
          			xStartMainPrc:=FALSE;
				xInitStep:=FALSE;
				(*10.09.2010: KFS	} *)
			END_IF;
		100:	xSetEndPrc:=FALSE;
			xStartMainPrc:=FALSE;
			xInitStep:=FALSE;
		(*SOA 27.02.23 *)
			T_ExchgParam.T_StationCommon.T_AutoGeometryPara.xMoveTableStuderBW := TRUE; (*Move Table Backwards*)
			TONStartTimer2(IN:=TRUE,PT:=T#2s);
				IF TONStartTimer2.Q THEN
					TONStartTimer2(IN:=FALSE);
					iStepPrc:=0;
					xSetEnd:=TRUE;
				END_IF;
		(*SOA 27.02.23 *)
 	END_CASE;
END_IF;
(******************************************************************************************************************************************)
(****************************				             	Init / Reset Part                                                   *****************************)
(******************************************************************************************************************************************)
IF xSetEnd THEN
	xEnd:=TRUE;
	xInitStep:=FALSE;
	xSetEnd:=FALSE;
	xStop:=FALSE;
	xStartMainPrc:=FALSE;
	xTmpStop:=FALSE;
	xInitMainCtr:=FALSE;
	xStartMainCtr:=FALSE;
	xStart:=FALSE;
	xSetError:=FALSE;
	xQuitErr:=FALSE;
	xError:=FALSE;
	diErrorNr:=0;
	xInitError:=FALSE;
	xFreeze:=FALSE;
	xAbord:=FALSE;
	xTmpAbord:=FALSE;
	xSetEndPrc:=FALSE;
	xStartProcess:=FALSE;
	xDoNotMoveGrindPosition:=FALSE;
	T_ExchgParam.T_StationCommon.T_AutoGroovePara.xBlockGrindFeeder:=xDoNotMoveGrindPosition;
	iNumberOfGrooves:=1;
	T_ExchgParam.T_StationCommon.T_AutoGeometryPara.xMoveTableStuderBW := FALSE;
END_IF;
END_FUNCTION_BLOCK

(* POU PRG_PROCESS_LAYER4/FB_PROCESS/FB_PrcToolCalibration, ST *)
FUNCTION_BLOCK FB_PrcToolCalibration
VAR_INPUT
	xMicroRodActive: BOOL;				(* choice of the machine MicroWire or MicroRod *)
	xBeckhoffDriveActive: BOOL;			(* choice of the axis Beckhoff or EcoStep *)
	T_NovRAMData:ST_DATA_RETAIN;	(* Novram structure for all Machine parameter *)
END_VAR
VAR_IN_OUT
	xStart : BOOL;							(* start a process *)
	xStop : BOOL;							(* stop a process *)
	xQuitErr : BOOL;						(* quit an error *)
	xAbord : BOOL;						(* abord a process *)
	T_Station : ST_STATION;				(* data structure of the stationlevel *)
	T_Process : ST_PROCESS;			(* data strucuture of the processlevel *)
	xReset : BOOL;						(* reset the FB *)
	T_ExchgParam:ST_QVIS_EXCHG_PARAM;	(* data structure of the visualisation *)
END_VAR
VAR_OUTPUT
	xEnd : BOOL;							(* Endflag of the process *)
	xError : BOOL;							(* Errorflag of the process *)
	diErrorNr : DINT;						(* Error number of the process *)
END_VAR
VAR
	iStepPrc: INT;
	xInitStep: BOOL;
	xSetError: BOOL;
	xSetEnd: BOOL;
	xStartMainCtr: BOOL;
	xStartMainPrc: BOOL;
	xInitMainCtr: BOOL;
	xFreeze: BOOL;
	xInitError: BOOL;
	iStepError: INT;
	xTmpStop: BOOL;
	xSetTmpError: BOOL;
	xTmpAbord: BOOL;
	diTmpErrNr: DINT;
	xSetEndPrc : BOOL;
	iTmpFunctionNr:INT;
	xStopFctStation1: BOOL;
	iStepStop: INT;
	iTmpStationFunctionNr: INT;
	xStartProcess: BOOL;
	TONStartTimer: TON;
	tStepTime: TIME;
	TONStartTimer1: TON;
END_VAR
(****************************************************************************************************************************************************)
(***********                                      This Functionblock define the process for the ToolCalibration                                                  ************)
(****************************************************************************************************************************************************)

(******************************************************************************************************************************************)
(****************************				           Reset Function Part                                                 *****************************)
(******************************************************************************************************************************************)
IF xReset THEN
	xReset:=FALSE;
	xSetEnd:=TRUE;
END_IF;
(******************************************************************************************************************************************)
(****************************				              Error Controlling Part                                            *****************************)
(******************************************************************************************************************************************)
IF (xSetError OR T_Station.TControl.xError) AND NOT(xSetEnd) THEN
	IF NOT(xInitError) THEN
		iStepError:=100;
		xInitError:=TRUE;
		IF NOT(xSetError) THEN
			xSetError:=TRUE;
			xSetTmpError:=FALSE;
		ELSE
			xSetTmpError:=TRUE;
		END_IF;
	END_IF;
	CASE iStepError OF
		100:	IF T_Station.TControl.xError THEN
				diErrorNr:=T_Station.TControl.diErrorNr;
			END_IF;
			IF xSetTmpError THEN
				diErrorNr:=diTmpErrNr;
			END_IF;
			iStepError:=200;
		200:	IF xSetTmpError THEN
				xSetTmpError:=FALSE;
				xStopFctStation1:=FALSE;
				iStepError:=300;
			ELSE
				IF NOT(T_Station.TControl.xError) AND NOT(T_Station.TControl.xEnd) THEN
					IF (T_Station.TControl.iFunctNr = 1) THEN
						T_Station.TControl.xStop:=TRUE;
						xStopFctStation1:=TRUE;
					ELSE
						xStopFctStation1:=FALSE;
					END_IF;
				END_IF;
				iStepError:=300;
			END_IF;
		300:	IF xStopFctStation1 THEN
				IF NOT(T_Station.TControl.xStop) THEN
					xStopFctStation1:=FALSE;
				END_IF;
			END_IF;
			IF NOT(xStopFctStation1) THEN
				xError:=TRUE;
				iStepError:=400;
			END_IF;
		400:	IF xQuitErr THEN
				T_Station.TControl.xQuitError:=T_Station.TControl.xError;
				iStepError:=500;
			END_IF;
		500: IF NOT(T_Station.TControl.xQuitError) THEN
				xSetEnd:=TRUE;
			END_IF;
	END_CASE;
END_IF;
(******************************************************************************************************************************************)
(****************************				              Main Controlling Part                                            *****************************)
(******************************************************************************************************************************************)
IF (xStart OR xStartMainCtr) AND NOT(xSetEnd) AND NOT(xSetError) THEN
	IF NOT (xInitMainCtr) THEN
		iStepPrc:=10;
		xInitMainCtr:=TRUE;
		xStartMainCtr:=TRUE;
		xStart:=FALSE;
		xEnd:=FALSE;
		xSetEndPrc:=FALSE;
		iTmpFunctionNr:=1;
		xAbord:=FALSE;
		T_ExchgParam.T_InfoValueCommon.rActualWireFeedPosition:=0.0;
		T_ExchgParam.T_InfoValueCommon.rActualWireFeedSpeed:=0.0;
	END_IF;
	IF xStop AND NOT(xTmpStop) THEN
		xTmpStop:=TRUE;
		iStepStop:=1;
	END_IF;
	IF xTmpStop THEN
		CASE iStepStop OF
		1:	IF NOT(T_Station.TControl.xEnd) THEN
				T_Station.TControl.xStop:=TRUE;
				iStepStop:=10;
			ELSE
				iStepStop:=20;
			END_IF;
		10:	IF NOT(T_Station.TControl.xStop) THEN
				iStepStop:=20;
			END_IF;
		20:	IF NOT(T_Station.TControl.xStart) AND T_Station.TControl.xEnd THEN
				T_Station.TControl.iFunctNr:=4;
				T_Station.TControl.xStart:=TRUE;
				T_Station.THardware.TAxisGrindFeeder.T_CtrleSingle.lrAcceleration:=T_NovRAMData.T_Standard.T_TeachINGrindFeeder.rAcceleration;
				T_Station.THardware.TAxisGrindFeeder.T_CtrleSingle.lrDecceleration:=T_NovRAMData.T_Standard.T_TeachINGrindFeeder.rDeceleration;
				T_Station.THardware.TAxisGrindFeeder.T_CtrleSingle.lrPosition:=	T_NovRAMData.T_ProcessImageData.T_ProcessPara.rToolDiameterProcess +
																			T_NovRAMData.T_ProcessImageData.T_ProcessPara.rSecurityPosGrindFeedProcess;
				T_Station.THardware.TAxisGrindFeeder.T_CtrleSingle.lrVelocity:=T_NovRAMData.T_ProcessImageData.T_ProcessPara.rSpeedBackwardGrindFeed;
				iStepStop:=30;
			END_IF;
		(* Check Active Movement of the Axis *)
		30:	IF NOT(T_Station.TControl.xStart) AND T_Station.TControl.xEnd THEN
				T_Station.TControl.iFunctNr:=18;	(* Check Axis Movement, and stop it if moves *)
				T_Station.TControl.xStart:=TRUE;
				iStepStop:=40;
			END_IF;
		40:	IF NOT(T_Station.TControl.xStart) AND T_Station.TControl.xEnd THEN
				xStartMainPrc:=FALSE;
				xInitStep:=FALSE;
				iStepPrc:=0;
				xSetEnd:=TRUE;
				RETURN;
			END_IF;
		END_CASE;
		RETURN;
	END_IF;
	IF NOT(xStartMainPrc) THEN
		xStartMainPrc:=TRUE;
	END_IF;
END_IF;
(******************************************************************************************************************************************)
(****************************				             Main Procedure Part                                             *****************************)
(******************************************************************************************************************************************)
IF xStartProcess THEN
	TONStartTimer(IN:=TRUE,PT:=T#1s);
	IF TONStartTimer.Q THEN
		TONStartTimer(IN:=FALSE);
		IF (T_ExchgParam.T_InfoValueCommon.tAutoTimeLeft >= T#1s) THEN
			T_ExchgParam.T_InfoValueCommon.tAutoTimeLeft:=T_ExchgParam.T_InfoValueCommon.tAutoTimeLeft - T#1s;
		ELSE
			T_ExchgParam.T_InfoValueCommon.tAutoTimeLeft:=T#0s;
		END_IF;
	END_IF;
	tStepTime:=T_ExchgParam.T_InfoValueCommon.tAutoTimeTotal / 100;
	TONStartTimer1(IN:=TRUE,PT:=tStepTime);
	IF TONStartTimer1.Q THEN
		TONStartTimer1(IN:=FALSE);
		T_ExchgParam.T_InfoValueCommon.bProgressbarToolCalibration:=T_ExchgParam.T_InfoValueCommon.bProgressbarToolCalibration + 1;
		IF (T_ExchgParam.T_InfoValueCommon.bProgressbarToolCalibration >= 100) THEN
			T_ExchgParam.T_InfoValueCommon.bProgressbarToolCalibration:=100;
		END_IF;
	END_IF;
ELSE
	TONStartTimer(IN:=FALSE);
	TONStartTimer1(IN:=FALSE);
END_IF;
IF xStartMainPrc AND NOT(xSetEnd) AND NOT(xSetError) THEN
	CASE iStepPrc OF
		(* Check first if the ToolCalibration is available to start it *)
		10:	T_Station.THardware.TAxisToolLeft.T_CtrleSingle.lrAcceleration:=T_NovRAMData.T_Standard.T_TeachINToolLeft.rAcceleration;
			T_Station.THardware.TAxisToolLeft.T_CtrleSingle.lrDecceleration:=T_NovRAMData.T_Standard.T_TeachINToolLeft.rDeceleration;
			T_Station.THardware.TAxisToolCenter.T_CtrleSingle.lrAcceleration:=T_NovRAMData.T_Standard.T_TeachINToolCenter.rAcceleration;
			T_Station.THardware.TAxisToolCenter.T_CtrleSingle.lrDecceleration:=T_NovRAMData.T_Standard.T_TeachINToolCenter.rDeceleration;
			T_Station.THardware.TAxisToolRight.T_CtrleSingle.lrAcceleration:=T_NovRAMData.T_Standard.T_TeachINToolRight.rAcceleration;
			T_Station.THardware.TAxisToolRight.T_CtrleSingle.lrDecceleration:=T_NovRAMData.T_Standard.T_TeachINToolRight.rDeceleration;
			T_Station.THardware.TAxisToolFeeder.T_CtrleSingle.lrAcceleration:=T_NovRAMData.T_Standard.T_TeachINToolFeeder.rAcceleration;
			T_Station.THardware.TAxisToolFeeder.T_CtrleSingle.lrDecceleration:=T_NovRAMData.T_Standard.T_TeachINToolFeeder.rDeceleration;
			T_Station.THardware.TAxisGrindFeeder.T_CtrleSingle.lrAcceleration:=T_NovRAMData.T_Standard.T_TeachINGrindFeeder.rAcceleration;
			T_Station.THardware.TAxisGrindFeeder.T_CtrleSingle.lrDecceleration:=T_NovRAMData.T_Standard.T_TeachINGrindFeeder.rDeceleration;
			(* Only for MicroRod, check if the tool is clamped *)
			IF xMicroRodActive THEN
				(*22.12.2009: KFS	{ *)
				(*
				IF T_Station.THardware.TCylToolTension.T_CtrleCyl.xStatePosOn THEN
					xSetError:=TRUE;
					diTmpErrNr:=2;			(* Tool is not clamped *)
				END_IF;
				*)
				(*Added control if all cylinder for the tool are activated*)
				IF T_Station.THardware.TCylToolTension.T_CtrleCyl.xStatePosOn OR
				     T_Station.THardware.TCylToolLeftActive.T_CtrleCyl.T_Standard.xActivOn OR
 				     T_Station.THardware.TCylToolRightActive.T_CtrleCyl.T_Standard.xActivOn  OR
				   (* T_Station.THardware.TCylToolCenterActive.T_CtrleCyl.T_Standard.xActivOn OR*)	(* IGS auskommentiert, diesen Zyl gibts auf der M3 nicht *)
				     NOT(T_Station.THardware.TCylToolPrismaLeftActive.T_CtrleCyl.T_Standard.xActivOn) OR
				     NOT(T_Station.THardware.TCylToolPrismaRightActive.T_CtrleCyl.T_Standard.xActivOn) 	THEN
					xSetError:=TRUE;
					diTmpErrNr:=2;			(* Tool is not clamped *)
				END_IF;
				(*22.12.2009: KFS	} *)
			END_IF;
			(* Only for MicroRod, check if the Machine is referenced *)
			IF xMicroRodActive THEN
				IF NOT(T_Station.TControl.xReferenced) THEN
					xSetError:=TRUE;
					diTmpErrNr:=1;	(* Machine is not referenced *)
					RETURN;
				END_IF;
			END_IF;
			xStartMainPrc:=FALSE;
			xInitStep:=FALSE;
			iStepPrc:=11;
		(* Set the ToolTension force *)
		11:	IF NOT(xInitStep) THEN
				xInitStep:=TRUE;
				T_Station.THardware.TCylToolTension.T_CtrleCyl.iFunction:=2;	(* activate the ToolTension *)
				T_Station.THardware.TCylToolTension.T_CtrleCyl.T_AnalogCylinder.rForceIn:=T_NovRAMData.T_ProcessImageData.T_ProcessPara.rToolTensionProcess;
				IF xMicroRodActive THEN
					T_Station.THardware.TCylToolTension.T_Config.tDelayOn:=T#1s;
				ELSE
					T_Station.THardware.TCylToolTension.T_Config.tDelayOn:=T#0s;
				END_IF;
				T_Station.THardware.TCylToolTension.T_CtrleCyl.xExecute:=TRUE;
			END_IF;
			IF NOT(T_Station.THardware.TCylToolTension.T_CtrleCyl.xExecute) AND T_Station.THardware.TCylToolTension.T_CtrleCyl.xDone THEN
				(* Only for MicroRod, check if the tool is clamped *)
				IF xMicroRodActive THEN
					IF T_Station.THardware.TCylToolTension.T_CtrleCyl.xStatePosOn THEN
						xSetError:=TRUE;
						diTmpErrNr:=2;			(* Tool is not clamped *)
						RETURN;
					END_IF;
				END_IF;
				iStepPrc:=20;
				xStartMainPrc:=FALSE;
				xInitStep:=FALSE;
			END_IF;
		(* Switch First all Axis the power supply on *)
		20:	IF NOT(xInitStep) THEN
				xInitStep:=TRUE;
				T_Station.TControl.iFunctNr:=16;
				T_Station.TControl.xStart:=TRUE;
			END_IF;
			IF NOT(T_Station.TControl.xStart) AND T_Station.TControl.xEnd THEN
				iStepPrc:=30;
				xStartMainPrc:=FALSE;
				xInitStep:=FALSE;
				iTmpStationFunctionNr:=6;
				T_Station.THardware.TAxisToolLeft.T_CtrleSingle.rSetPosition:=0.0;
				T_Station.THardware.TAxisToolCenter.T_CtrleSingle.rSetPosition:=0.0;
				T_Station.THardware.TAxisToolRight.T_CtrleSingle.rSetPosition:=0.0;
				T_Station.THardware.TAxisToolFeeder.T_CtrleSingle.rSetPosition:=0.0;
			END_IF;
		(* Reset the Position of the Axis *)
		30:	IF NOT(xInitStep) THEN
				xInitStep:=TRUE;
				(* 6=ToolLeft, 7=ToolCenter, 8=ToolRight, 9=ToolFeeder *)
				T_Station.TControl.iFunctNr:=iTmpStationFunctionNr;
				T_Station.TControl.xStart:=TRUE;
			END_IF;
			IF NOT(T_Station.TControl.xStart) AND T_Station.TControl.xEnd THEN
				iTmpStationFunctionNr:=iTmpStationFunctionNr + 1;
				IF NOT(xMicroRodActive) AND (iTmpStationFunctionNr = 7) THEN
					iTmpStationFunctionNr:=iTmpStationFunctionNr + 1;
				END_IF;
				IF xMicroRodActive AND (iTmpStationFunctionNr = 9) THEN
					iTmpStationFunctionNr:=iTmpStationFunctionNr + 1;
				END_IF;
				xStartMainPrc:=FALSE;
				xInitStep:=FALSE;
				IF (iTmpStationFunctionNr < 10) THEN
					iStepPrc:=30;
				ELSE
					iStepPrc:=40;
				END_IF;
			END_IF;
		(* GrindFeeder Set Absolut to Security Position *)
		40:	IF NOT(xInitStep) THEN
				xInitStep:=TRUE;
				T_Station.TControl.iFunctNr:=4;
				T_Station.TControl.xStart:=TRUE;
				T_Station.THardware.TAxisGrindFeeder.T_CtrleSingle.lrAcceleration:=T_NovRAMData.T_Standard.T_TeachINGrindFeeder.rAcceleration;
				T_Station.THardware.TAxisGrindFeeder.T_CtrleSingle.lrDecceleration:=T_NovRAMData.T_Standard.T_TeachINGrindFeeder.rDeceleration;
				T_Station.THardware.TAxisGrindFeeder.T_CtrleSingle.lrPosition:=	T_NovRAMData.T_ProcessImageData.T_ProcessPara.rToolDiameterProcess +
																			T_NovRAMData.T_ProcessImageData.T_ProcessPara.rSecurityPosGrindFeedProcess;
				T_Station.THardware.TAxisGrindFeeder.T_CtrleSingle.lrVelocity:=T_NovRAMData.T_ProcessImageData.T_ProcessPara.rSpeedBackwardGrindFeed;
			END_IF;
			IF NOT(T_Station.TControl.xStart) AND T_Station.TControl.xEnd THEN
				IF xMicroRodActive THEN
					iStepPrc:=50;
				ELSE
					iStepPrc:=60;
				END_IF;
				xStartMainPrc:=FALSE;
				xInitStep:=FALSE;
			END_IF;
		(* Only for MicroRod-->Set ToolFeed Absolut to the StartPosition and if more cycle than only the first time *)
		50:	IF NOT(xInitStep) THEN
				xInitStep:=TRUE;
				T_Station.TControl.iFunctNr:=14;
				T_Station.TControl.xStart:=TRUE;
				T_Station.THardware.TAxisToolFeeder.T_CtrleSingle.lrAcceleration:=T_NovRAMData.T_Standard.T_TeachINToolFeeder.rAcceleration;
				T_Station.THardware.TAxisToolFeeder.T_CtrleSingle.lrDecceleration:=T_NovRAMData.T_Standard.T_TeachINToolFeeder.rDeceleration;
				T_Station.THardware.TAxisToolFeeder.T_CtrleSingle.lrPosition:=T_NovRAMData.T_ProcessImageData.T_CalibrationPara.rStartPosToolFeedCalib;
				T_Station.THardware.TAxisToolFeeder.T_CtrleSingle.lrVelocity:=T_NovRAMData.T_ProcessImageData.T_ProcessPara.rSpeedStartPosToolFeedProcess;
			END_IF;
			IF NOT(T_Station.TControl.xStart) AND T_Station.TControl.xEnd THEN
				iStepPrc:=60;
				xStartMainPrc:=FALSE;
				xInitStep:=FALSE;
			END_IF;
		(* ToolRotation Start *)
		60:	IF NOT(xInitStep) THEN
				xInitStep:=TRUE;
				T_Station.TControl.iFunctNr:=2;
				T_Station.TControl.xStart:=TRUE;
				(* ToolLeft --> Master *)
				T_Station.THardware.TAxisToolLeft.T_CtrleSingle.lrVelocity:=T_NovRAMData.T_ProcessImageData.T_CalibrationPara.rSpeedToolRotationCalib;
				T_Station.THardware.TAxisToolLeft.T_CtrleSingle.lrAcceleration:=T_NovRAMData.T_Standard.T_TeachINToolLeft.rAcceleration;
				T_Station.THardware.TAxisToolLeft.T_CtrleSingle.lrDecceleration:=T_NovRAMData.T_Standard.T_TeachINToolLeft.rDeceleration;
				IF xMicroRodActive THEN
					(* ToolCenter --> Slave of ToolLeft only by MicroRod *)
					T_Station.THardware.TAxisToolCenter.T_CtrleSingle.lrAcceleration:=T_NovRAMData.T_Standard.T_TeachINToolCenter.rAcceleration;
					T_Station.THardware.TAxisToolCenter.T_CtrleSingle.lrDecceleration:=T_NovRAMData.T_Standard.T_TeachINToolCenter.rDeceleration;
					T_Station.THardware.TAxisToolCenter.T_CtrleSingle.lrGearDivider:=INT_TO_LREAL(T_Station.T_WorkTool.iBaseGearDivider);
					T_Station.THardware.TAxisToolCenter.T_CtrleSingle.lrGearFactor:=(	INT_TO_LREAL(T_Station.T_WorkTool.iBaseGearDivider) /
																					(T_Station.THardware.TAxisToolLeft.T_CtrleSingle.lrGearRatio /
																					T_Station.THardware.TAxisToolCenter.T_CtrleSingle.lrGearRatio)) * -1.0;

					(* ToolRight --> Slave of ToolLeft by MicroWire or Slave of ToolRight by MicroRod *)
					T_Station.THardware.TAxisToolRight.T_CtrleSingle.lrAcceleration:=T_NovRAMData.T_Standard.T_TeachINToolRight.rAcceleration;
					T_Station.THardware.TAxisToolRight.T_CtrleSingle.lrDecceleration:=T_NovRAMData.T_Standard.T_TeachINToolRight.rDeceleration;
					T_Station.THardware.TAxisToolRight.T_CtrleSingle.lrGearDivider:=INT_TO_LREAL(T_Station.T_WorkTool.iBaseGearDivider);
					T_Station.THardware.TAxisToolRight.T_CtrleSingle.lrGearFactor:=	INT_TO_LREAL(T_Station.T_WorkTool.iBaseGearDivider) /
																					(T_Station.THardware.TAxisToolLeft.T_CtrleSingle.lrGearRatio /
																					T_Station.THardware.TAxisToolRight.T_CtrleSingle.lrGearRatio);
				END_IF;

				IF NOT(xMicroRodActive) THEN
					(* ToolRight --> Slave of ToolRight by MicroWire *)
					T_Station.THardware.TAxisToolFeeder.T_CtrleSingle.lrAcceleration:=T_NovRAMData.T_Standard.T_TeachINToolFeeder.rAcceleration;
					T_Station.THardware.TAxisToolFeeder.T_CtrleSingle.lrDecceleration:=T_NovRAMData.T_Standard.T_TeachINToolFeeder.rDeceleration;
					T_Station.THardware.TAxisToolFeeder.T_CtrleSingle.lrGearDivider:=INT_TO_LREAL(T_Station.T_WorkTool.iBaseGearDivider);
					T_Station.THardware.TAxisToolFeeder.T_CtrleSingle.lrGearFactor:=	(INT_TO_LREAL(T_Station.T_WorkTool.iBaseGearDivider) /
																					(T_Station.THardware.TAxisToolFeeder.T_CtrleSingle.lrGearRatio /
																					T_Station.THardware.TAxisToolRight.T_CtrleSingle.lrGearRatio)) * -1.0;

					(* ToolRight --> Slave of ToolLeft by MicroWire or Slave of ToolRight by MicroRod *)
					T_Station.THardware.TAxisToolRight.T_CtrleSingle.lrAcceleration:=T_NovRAMData.T_Standard.T_TeachINToolRight.rAcceleration;
					T_Station.THardware.TAxisToolRight.T_CtrleSingle.lrDecceleration:=T_NovRAMData.T_Standard.T_TeachINToolRight.rDeceleration;
					T_Station.THardware.TAxisToolRight.T_CtrleSingle.lrGearDivider:=INT_TO_LREAL(T_Station.T_WorkTool.iBaseGearDivider);
					T_Station.THardware.TAxisToolRight.T_CtrleSingle.lrGearFactor:=	(INT_TO_LREAL(T_Station.T_WorkTool.iBaseGearDivider) /
																					(T_Station.THardware.TAxisToolLeft.T_CtrleSingle.lrGearRatio /
																					T_Station.THardware.TAxisToolRight.T_CtrleSingle.lrGearRatio)) * -1.0;
				END_IF;
			END_IF;
			IF NOT(T_Station.TControl.xStart) AND T_Station.TControl.xEnd THEN
				xStartMainPrc:=FALSE;
				xInitStep:=FALSE;
				iStepPrc:=70;
			END_IF;
		(* GrindFeeder Set Absolut to ToolDiameter minus the offset with the fast speed *)
		70:	IF NOT(xInitStep) THEN
				xInitStep:=TRUE;
				T_Station.TControl.iFunctNr:=4;
				T_Station.TControl.xStart:=TRUE;
				T_Station.THardware.TAxisGrindFeeder.T_CtrleSingle.lrAcceleration:=T_NovRAMData.T_Standard.T_TeachINGrindFeeder.rAcceleration;
				T_Station.THardware.TAxisGrindFeeder.T_CtrleSingle.lrDecceleration:=T_NovRAMData.T_Standard.T_TeachINGrindFeeder.rDeceleration;
				T_Station.THardware.TAxisGrindFeeder.T_CtrleSingle.lrPosition:=T_NovRAMData.T_ProcessImageData.T_ProcessPara.rToolDiameterProcess + T_NovRAMData.T_ProcessImageData.T_ProcessPara.rOffsetBeforeToolDiaGrindFeedProcess;
				T_Station.THardware.TAxisGrindFeeder.T_CtrleSingle.lrVelocity:=T_NovRAMData.T_ProcessImageData.T_ProcessPara.rSpeedForwardFastGrindFeed;
			END_IF;
			IF NOT(T_Station.TControl.xStart) AND T_Station.TControl.xEnd THEN
				xStartMainPrc:=FALSE;
				xInitStep:=FALSE;
				iStepPrc:=80;
			END_IF;
		(* Working ToolCalibration *)
		80:	IF NOT(xInitStep) THEN
				xStartProcess:=TRUE;
				xInitStep:=TRUE;
				T_Station.TControl.iFunctNr:=13;
				T_Station.TControl.xStart:=TRUE;
			END_IF;
			IF NOT(T_Station.TControl.xStart) AND T_Station.TControl.xEnd THEN
				xStartMainPrc:=FALSE;
				xInitStep:=FALSE;
				iStepPrc:=90;
				RETURN;
			END_IF;
			(* Only for MicroRod, check if the tool is clamped *)
			IF xMicroRodActive THEN
				IF T_Station.THardware.TCylToolTension.T_CtrleCyl.xStatePosOn THEN
					xStartMainPrc:=FALSE;
					xInitStep:=FALSE;
					iStepPrc:=81;
					RETURN;
				END_IF;
			END_IF;
		(* Stop the Process, because the Tool is broken *)
		81:	IF NOT(xInitStep) THEN
				xInitStep:=TRUE;
				T_Station.TControl.xStop:=TRUE;
			END_IF;
			IF NOT(T_Station.TControl.xStart) AND T_Station.TControl.xEnd THEN
				xStartMainPrc:=FALSE;
				xInitStep:=FALSE;
				iStepPrc:=82;
			END_IF;
		(* Set the GrindFeeder to the security Position *)
		82:	IF NOT(xInitStep) THEN
				xInitStep:=TRUE;
				T_Station.TControl.iFunctNr:=4;
				T_Station.TControl.xStart:=TRUE;
				T_Station.THardware.TAxisGrindFeeder.T_CtrleSingle.lrAcceleration:=T_NovRAMData.T_Standard.T_TeachINGrindFeeder.rAcceleration;
				T_Station.THardware.TAxisGrindFeeder.T_CtrleSingle.lrDecceleration:=T_NovRAMData.T_Standard.T_TeachINGrindFeeder.rDeceleration;
				T_Station.THardware.TAxisGrindFeeder.T_CtrleSingle.lrPosition:=	T_NovRAMData.T_ProcessImageData.T_ProcessPara.rToolDiameterProcess +
																			T_NovRAMData.T_ProcessImageData.T_ProcessPara.rSecurityPosGrindFeedProcess;
				T_Station.THardware.TAxisGrindFeeder.T_CtrleSingle.lrVelocity:=T_NovRAMData.T_ProcessImageData.T_ProcessPara.rSpeedBackwardGrindFeed;
			END_IF;
			IF NOT(T_Station.TControl.xStart) AND T_Station.TControl.xEnd THEN
				xStartMainPrc:=FALSE;
				xInitStep:=FALSE;
				iStepPrc:=83;
			END_IF;
		(* Check Active Movement of the Axis *)
		83:	IF NOT(xInitStep) THEN
				xInitStep:=TRUE;
				T_Station.TControl.iFunctNr:=18;	(* Check Axis Movement, and stop it if moves *)
				T_Station.TControl.xStart:=TRUE;
			END_IF;
			IF NOT(T_Station.TControl.xStart) AND T_Station.TControl.xEnd THEN
				xSetError:=TRUE;
				diTmpErrNr:=2;			(* Tool is not clamped *)
				RETURN;
			END_IF;
		(* GrindFeeder Set Absolut to Security Position *)
		90:	IF NOT(xInitStep) THEN
				xInitStep:=TRUE;
				T_Station.TControl.iFunctNr:=4;
				T_Station.TControl.xStart:=TRUE;
				T_Station.THardware.TAxisGrindFeeder.T_CtrleSingle.lrAcceleration:=T_NovRAMData.T_Standard.T_TeachINGrindFeeder.rAcceleration;
				T_Station.THardware.TAxisGrindFeeder.T_CtrleSingle.lrDecceleration:=T_NovRAMData.T_Standard.T_TeachINGrindFeeder.rDeceleration;
				T_Station.THardware.TAxisGrindFeeder.T_CtrleSingle.lrPosition:=	T_NovRAMData.T_ProcessImageData.T_ProcessPara.rToolDiameterProcess +
																			T_NovRAMData.T_ProcessImageData.T_ProcessPara.rSecurityPosGrindFeedProcess;
				T_Station.THardware.TAxisGrindFeeder.T_CtrleSingle.lrVelocity:=T_NovRAMData.T_ProcessImageData.T_ProcessPara.rSpeedBackwardGrindFeed;
			END_IF;
			IF NOT(T_Station.TControl.xStart) AND T_Station.TControl.xEnd THEN
				xStartMainPrc:=FALSE;
				xInitStep:=FALSE;
				iStepPrc:=100;
			END_IF;
		(* ToolRotation Stop *)
		100:	IF NOT(xInitStep) THEN
				xInitStep:=TRUE;
				T_Station.TControl.iFunctNr:=3;
				T_Station.TControl.xStart:=TRUE;
				(* ToolLeft --> Master *)
				T_Station.THardware.TAxisToolLeft.T_CtrleSingle.lrAcceleration:=T_NovRAMData.T_Standard.T_TeachINToolLeft.rAcceleration;
				T_Station.THardware.TAxisToolLeft.T_CtrleSingle.lrDecceleration:=T_NovRAMData.T_Standard.T_TeachINToolLeft.rDeceleration;
				IF xMicroRodActive THEN
					(* ToolCenter --> Slave of ToolLeft only by MicroRod *)
					T_Station.THardware.TAxisToolCenter.T_CtrleSingle.lrAcceleration:=T_NovRAMData.T_Standard.T_TeachINToolCenter.rAcceleration;
					T_Station.THardware.TAxisToolCenter.T_CtrleSingle.lrDecceleration:=T_NovRAMData.T_Standard.T_TeachINToolCenter.rDeceleration;
				END_IF;
				(* ToolRight --> Slave of ToolLeft by MicroWire or Slave of ToolRight by MicroRod *)
				T_Station.THardware.TAxisToolRight.T_CtrleSingle.lrAcceleration:=T_NovRAMData.T_Standard.T_TeachINToolRight.rAcceleration;
				T_Station.THardware.TAxisToolRight.T_CtrleSingle.lrDecceleration:=T_NovRAMData.T_Standard.T_TeachINToolRight.rDeceleration;
				IF NOT(xMicroRodActive) THEN
					(* ToolRight --> Slave of ToolRight by MicroWire *)
					T_Station.THardware.TAxisToolFeeder.T_CtrleSingle.lrAcceleration:=T_NovRAMData.T_Standard.T_TeachINToolFeeder.rAcceleration;
					T_Station.THardware.TAxisToolFeeder.T_CtrleSingle.lrDecceleration:=T_NovRAMData.T_Standard.T_TeachINToolFeeder.rDeceleration;
				END_IF;
			END_IF;
			IF NOT(T_Station.TControl.xStart) AND T_Station.TControl.xEnd THEN
				xStartMainPrc:=FALSE;
				xInitStep:=FALSE;
				iStepPrc:=110;
			END_IF;
		110:	xSetEndPrc:=FALSE;
			xStartMainPrc:=FALSE;
			xInitStep:=FALSE;
			iStepPrc:=0;
			xSetEnd:=TRUE;
	END_CASE;
END_IF;
(******************************************************************************************************************************************)
(****************************				             	Init / Reset Part                                                   *****************************)
(******************************************************************************************************************************************)
IF xSetEnd THEN
	xEnd:=TRUE;
	xInitStep:=FALSE;
	xSetEnd:=FALSE;
	xStop:=FALSE;
	xStartMainPrc:=FALSE;
	xTmpStop:=FALSE;
	xInitMainCtr:=FALSE;
	xStartMainCtr:=FALSE;
	xStart:=FALSE;
	xSetError:=FALSE;
	xQuitErr:=FALSE;
	xError:=FALSE;
	diErrorNr:=0;
	xInitError:=FALSE;
	xFreeze:=FALSE;
	xAbord:=FALSE;
	xTmpAbord:=FALSE;
	xSetEndPrc:=FALSE;
	xStartProcess:=FALSE;
END_IF;
END_FUNCTION_BLOCK

(* POU PRG_STATION_LAYER3/PRG_STATION, FBD *)
PROGRAM PRG_STATION
VAR
	FBStation: FB_STATION;
END_VAR
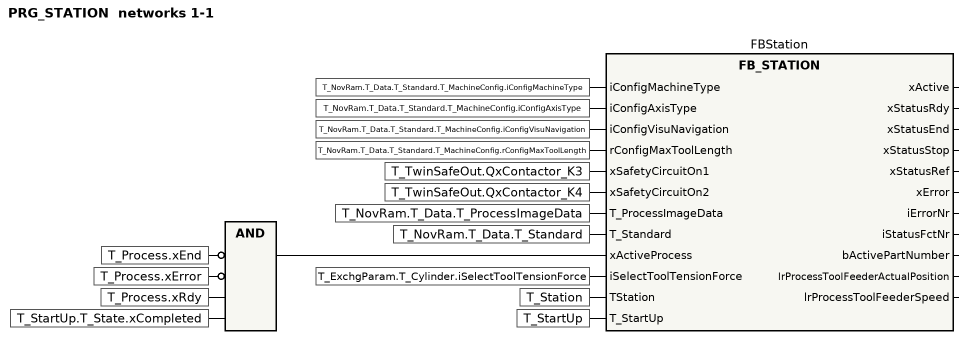
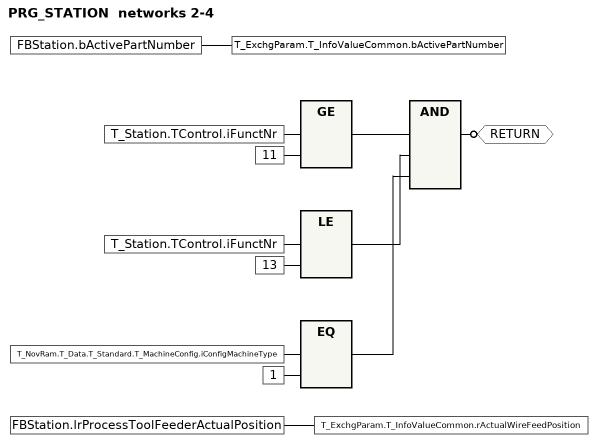
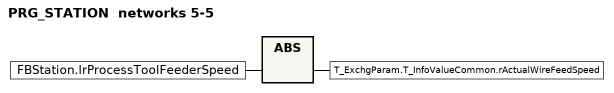
_FBD_ (* Function Block Diagram *)
NETWORK 1 (* STATION LEVEL-->LAYER 3 *)
	FBStation:FB_STATION(iConfigMachineType: T_NovRam.T_Data.T_Standard.T_MachineConfig.iConfigMachineType, iConfigAxisType: T_NovRam.T_Data.T_Standard.T_MachineConfig.iConfigAxisType, iConfigVisuNavigation: T_NovRam.T_Data.T_Standard.T_MachineConfig.iConfigVisuNavigation, rConfigMaxToolLength: T_NovRam.T_Data.T_Standard.T_MachineConfig.rConfigMaxToolLength, xSafetyCircuitOn1: T_TwinSafeOut.QxContactor_K3, xSafetyCircuitOn2: T_TwinSafeOut.QxContactor_K4, T_ProcessImageData: T_NovRam.T_Data.T_ProcessImageData, T_Standard: T_NovRam.T_Data.T_Standard, xActiveProcess: AND(NOT T_Process.xEnd, NOT T_Process.xError, T_Process.xRdy, T_StartUp.T_State.xCompleted), iSelectToolTensionForce: T_ExchgParam.T_Cylinder.iSelectToolTensionForce, TStation: T_Station, T_StartUp: T_StartUp)
NETWORK 2
	FBStation.bActivePartNumber => T_ExchgParam.T_InfoValueCommon.bActivePartNumber
NETWORK 3
	NOT AND(GE(T_Station.TControl.iFunctNr, 11), LE(T_Station.TControl.iFunctNr, 13), EQ(T_NovRam.T_Data.T_Standard.T_MachineConfig.iConfigMachineType, 1)) => <RETURN>
NETWORK 4
	FBStation.lrProcessToolFeederActualPosition => T_ExchgParam.T_InfoValueCommon.rActualWireFeedPosition
NETWORK 5
	ABS(FBStation.lrProcessToolFeederSpeed) => T_ExchgParam.T_InfoValueCommon.rActualWireFeedSpeed
_END_FBD_
(* the same logic as Structured Text *)
(* Network 1: STATION LEVEL-->LAYER 3 *)
FBStation(iConfigMachineType := T_NovRam.T_Data.T_Standard.T_MachineConfig.iConfigMachineType, iConfigAxisType := T_NovRam.T_Data.T_Standard.T_MachineConfig.iConfigAxisType, iConfigVisuNavigation := T_NovRam.T_Data.T_Standard.T_MachineConfig.iConfigVisuNavigation, rConfigMaxToolLength := T_NovRam.T_Data.T_Standard.T_MachineConfig.rConfigMaxToolLength, xSafetyCircuitOn1 := T_TwinSafeOut.QxContactor_K3, xSafetyCircuitOn2 := T_TwinSafeOut.QxContactor_K4, T_ProcessImageData := T_NovRam.T_Data.T_ProcessImageData, T_Standard := T_NovRam.T_Data.T_Standard, xActiveProcess := NOT T_Process.xEnd AND NOT T_Process.xError AND T_Process.xRdy AND T_StartUp.T_State.xCompleted, iSelectToolTensionForce := T_ExchgParam.T_Cylinder.iSelectToolTensionForce, TStation := T_Station, T_StartUp := T_StartUp);
(* Network 2 *)
T_ExchgParam.T_InfoValueCommon.bActivePartNumber := FBStation.bActivePartNumber;
(* Network 3 *)
IF NOT ((T_Station.TControl.iFunctNr >= 11) AND (T_Station.TControl.iFunctNr <= 13) AND (T_NovRam.T_Data.T_Standard.T_MachineConfig.iConfigMachineType = 1)) THEN RETURN; END_IF;
(* Network 4 *)
T_ExchgParam.T_InfoValueCommon.rActualWireFeedPosition := FBStation.lrProcessToolFeederActualPosition;
(* Network 5 *)
T_ExchgParam.T_InfoValueCommon.rActualWireFeedSpeed := ABS(FBStation.lrProcessToolFeederSpeed);
END_PROGRAM

